LIN {X 0,Y 361.89,Z 300.406,A -85,B 0,C 180,E1 -12980.461,E2 -12980.461} C_VEL
LIN {X 0,Y 361.897,Z 300.402,A -85,B 0,C 180,E1 -12984.112,E2 -12984.112} C_VEL
LIN {X 0,Y 361.838,Z 300.409,A -85,B 0,C 180,E1 -12987.785,E2 -12987.785} C_VEL
LIN {X 0,Y 361.848,Z 300.411,A -85,B 0,C 180,E1 -12991.284,E2 -12991.284} C_VEL
LIN {X 0,Y 361.854,Z 300.407,A -85,B 0,C 180,E1 -12994.28,E2 -12994.28} C_VEL
LIN {X 0,Y 361.861,Z 300.411,A -85,B 0,C 180,E1 -12997.221,E2 -12997.221} C_VEL
LIN {X 0,Y 361.814,Z 300.414,A -85,B 0,C 180,E1 -13000.75,E2 -13000.75} C_VEL
LIN {X 0,Y 361.814,Z 300.412,A -85,B 0,C 180,E1 -13004.369,E2 -13004.369} C_VEL
LIN {X 0,Y 361.831,Z 300.414,A -85,B 0,C 180,E1 -13007.569,E2 -13007.569} C_VEL
LIN {X 0,Y 361.845,Z 300.413,A -85,B 0,C 180,E1 -13011.571,E2 -13011.571} C_VEL
LIN {X 0,Y 361.872,Z 300.405,A -85,B 0,C 180,E1 -13014.656,E2 -13014.656} C_VEL
LIN {X 0,Y 361.84,Z 300.413,A -85,B 0,C 180,E1 -13018.37,E2 -13018.37} C_VEL
LIN {X 0,Y 361.91,Z 300.458,A -85,B 0,C 180,E1 -13020.35,E2 -13020.35} C_VEL
LIN {X 0,Y 364.458,Z 313.266,A -85,B 0,C 180,E1 -13023.398,E2 -13023.398} C_VEL
LIN {X 0,Y 365.319,Z 318.996,A -85,B 0,C 180,E1 -13024.714,E2 -13024.714} C_VEL
LIN {X 0,Y 363.817,Z 337.623,A -85,B 0,C 180,E1 -13028.704,E2 -13028.704} C_VEL
LIN {X 0,Y 368.558,Z 374.157,A -85,B 0,C 180,E1 -13029.685,E2 -13029.685} C_VEL
LIN {X 0,Y 367.481,Z 446.165,A -85,B 0,C 180,E1 -13031.099,E2 -13031.099} C_VEL
LIN {X 0,Y 366.821,Z 459.565,A -85,B 0,C 180,E1 -13031.57,E2 -13031.57} C_VEL
LIN {X 0,Y 366.07,Z 472.403,A -85,B 0,C 180,E1 -13032.255,E2 -13032.255} C_VEL
LIN {X 0,Y 365.162,Z 483.779,A -85,B 0,C 180,E1 -13033.076,E2 -13033.076} C_VEL
LIN {X 0,Y 364.124,Z 495.519,A -85,B 0,C 180,E1 -13034.179,E2 -13034.179} C_VEL
LIN {X 0,Y 363.263,Z 506.09,A -85,B 0,C 180,E1 -13035.432,E2 -13035.432} C_VEL
LIN {X 0,Y 362.404,Z 515.589,A -85,B 0,C 180,E1 -13036.828,E2 -13036.828} C_VEL
LIN {X 0,Y 361.739,Z 523.371,A -85,B 0,C 180,E1 -13038.228,E2 -13038.228} C_VEL
LIN {X 0,Y 361.12,Z 530.982,A -85,B 0,C 180,E1 -13039.912,E2 -13039.912} C_VEL
LIN {X 0,Y 360.705,Z 537.097,A -85,B 0,C 180,E1 -13041.597,E2 -13041.597} C_VEL
LIN {X 0,Y 360.497,Z 541.932,A -85,B 0,C 180,E1 -13043.282,E2 -13043.282} C_VEL
LIN {X 0,Y 360.413,Z 545.63,A -85,B 0,C 180,E1 -13044.965,E2 -13044.965} C_VEL
LIN {X 0,Y 360.342,Z 548.292,A -85,B 0,C 180,E1 -13046.645,E2 -13046.645} C_VEL
LIN {X 0,Y 360.39,Z 549.547,A -85,B 0,C 180,E1 -13047.764,E2 -13047.764} C_VEL
LIN {X 0,Y 360.474,Z 550.389,A -85,B 0,C 180,E1 -13048.882,E2 -13048.882} C_VEL
LIN {X 0,Y 360.478,Z 550.79,A -85,B 0,C 180,E1 -13049.999,E2 -13049.999} C_VEL
LIN {X 0,Y 360.453,Z 550.799,A -85,B 0,C 180,E1 -13051.116,E2 -13051.116} C_VEL
LIN {X 0,Y 360.324,Z 549.647,A -85,B 0,C 180,E1 -13053.354,E2 -13053.354} C_VEL
LIN {X 0,Y 360.368,Z 548.437,A -85,B 0,C 180,E1 -13054.473,E2 -13054.473} C_VEL
LIN {X 0,Y 360.377,Z 546.224,A -85,B 0,C 180,E1 -13055.96,E2 -13055.96} C_VEL
LIN {X 0,Y 360.658,Z 542.298,A -85,B 0,C 180,E1 -13057.839,E2 -13057.839} C_VEL
LIN {X 0,Y 361.037,Z 537.639,A -85,B 0,C 180,E1 -13059.523,E2 -13059.523} C_VEL
LIN {X 0,Y 361.794,Z 530.633,A -85,B 0,C 180,E1 -13061.484,E2 -13061.484} C_VEL
LIN {X 0,Y 362.831,Z 523.079,A -85,B 0,C 180,E1 -13063.155,E2 -13063.155} C_VEL
LIN {X 0,Y 363.926,Z 513.963,A -85,B 0,C 180,E1 -13064.773,E2 -13064.773} C_VEL
LIN {X 0,Y 365.164,Z 503.913,A -85,B 0,C 180,E1 -13066.204,E2 -13066.204} C_VEL
LIN {X 0,Y 366.504,Z 493.117,A -85,B 0,C 180,E1 -13067.434,E2 -13067.434} C_VEL
LIN {X 0,Y 367.68,Z 482.609,A -85,B 0,C 180,E1 -13068.384,E2 -13068.384} C_VEL
LIN {X 0,Y 368.89,Z 469.987,A -85,B 0,C 180,E1 -13069.258,E2 -13069.258} C_VEL
LIN {X 0,Y 369.903,Z 456.623,A -85,B 0,C 180,E1 -13069.925,E2 -13069.925} C_VEL
LIN {X 0,Y 370.552,Z 444.241,A -85,B 0,C 180,E1 -13070.32,E2 -13070.32} C_VEL
LIN {X 0,Y 371.853,Z 373.551,A -85,B 0,C 180,E1 -13071.717,E2 -13071.717} C_VEL
LIN {X 0,Y 368.117,Z 350.904,A -85,B 0,C 180,E1 -13072.459,E2 -13072.459} C_VEL
LIN {X 0,Y 365.404,Z 336.978,A -85,B 0,C 180,E1 -13072.983,E2 -13072.983} C_VEL
LIN {X 0,Y 366.681,Z 324.457,A -85,B 0,C 180,E1 -13075.733,E2 -13075.733} C_VEL
LIN {X 0,Y 366.508,Z 321.277,A -85,B 0,C 180,E1 -13076.476,E2 -13076.476} C_VEL
LIN {X 0,Y 364.106,Z 309.636,A -85,B 0,C 180,E1 -13079.4,E2 -13079.4} C_VEL
LIN {X 0,Y 361.877,Z 300.409,A -85,B 0,C 180,E1 -13081.87,E2 -13081.87} C_VEL
LIN {X 0,Y 361.865,Z 300.412,A -85,B 0,C 180,E1 -13085.636,E2 -13085.636} C_VEL
LIN {X 0,Y 361.865,Z 300.407,A -85,B 0,C 180,E1 -13089.026,E2 -13089.026} C_VEL
LIN {X 0,Y 361.833,Z 300.414,A -85,B 0,C 180,E1 -13092.828,E2 -13092.828} C_VEL
LIN {X 0,Y 361.815,Z 300.415,A -85,B 0,C 180,E1 -13095.946,E2 -13095.946} C_VEL
LIN {X 0,Y 361.833,Z 300.409,A -85,B 0,C 180,E1 -13099.244,E2 -13099.244} C_VEL
LIN {X 0,Y 361.86,Z 300.409,A -85,B 0,C 180,E1 -13102.777,E2 -13102.777} C_VEL
LIN {X 0,Y 361.85,Z 300.404,A -85,B 0,C 180,E1 -13105.719,E2 -13105.719} C_VEL
LIN {X 0,Y 361.869,Z 300.404,A -85,B 0,C 180,E1 -13109.672,E2 -13109.672} C_VEL
LIN {X 0,Y 361.95,Z 300.395,A -85,B 0,C 180,E1 -13113.475,E2 -13113.475} C_VEL
LIN {X 0,Y 361.888,Z 300.405,A -85,B 0,C 180,E1 -13117.145,E2 -13117.145} C_VEL
LIN {X 0,Y 361.903,Z 300.402,A -85,B 0,C 180,E1 -13120.723,E2 -13120.723} C_VEL
LIN {X 0,Y 361.929,Z 300.396,A -85,B 0,C 180,E1 -13123.066,E2 -13123.066} C_VEL
LIN {X 0,Y 361.995,Z 300.395,A -85,B 0,C 180,E1 -13126.528,E2 -13126.528} C_VEL
LIN {X 0,Y 362.028,Z 300.387,A -85,B 0,C 180,E1 -13129.938,E2 -13129.938} C_VEL
LIN {X 0,Y 362.147,Z 300.367,A -85,B 0,C 180,E1 -13132.193,E2 -13132.193} C_VEL
LIN {X 0,Y 362.115,Z 300.378,A -85,B 0,C 180,E1 -13134.431,E2 -13134.431} C_VEL
LIN {X 0,Y 362.28,Z 300.354,A -85,B 0,C 180,E1 -13137.777,E2 -13137.777} C_VEL
LIN {X 0,Y 362.425,Z 300.333,A -85,B 0,C 180,E1 -13140,E2 -13140} C_VEL
LIN {X 0,Y 362.279,Z 300.354,A -85,B 0,C 180,E1 -13142.224,E2 -13142.224} C_VEL
LIN {X 0,Y 362.169,Z 300.37,A -85,B 0,C 180,E1 -13146.687,E2 -13146.687} C_VEL
LIN {X 0,Y 362.071,Z 300.379,A -85,B 0,C 180,E1 -13148.934,E2 -13148.934} C_VEL
LIN {X 0,Y 361.957,Z 300.395,A -85,B 0,C 180,E1 -13152.333,E2 -13152.333} C_VEL
LIN {X 0,Y 361.959,Z 300.394,A -85,B 0,C 180,E1 -13154.621,E2 -13154.621} C_VEL
LIN {X 0,Y 361.953,Z 300.393,A -85,B 0,C 180,E1 -13158.1,E2 -13158.1} C_VEL
LIN {X 0,Y 361.889,Z 300.402,A -85,B 0,C 180,E1 -13161.654,E2 -13161.654} C_VEL
LIN {X 0,Y 361.926,Z 300.398,A -85,B 0,C 180,E1 -13165.291,E2 -13165.291} C_VEL
LIN {X 0,Y 361.906,Z 300.401,A -85,B 0,C 180,E1 -13167.78,E2 -13167.78} C_VEL
LIN {X 0,Y 361.835,Z 300.408,A -85,B 0,C 180,E1 -13171.63,E2 -13171.63} C_VEL
LIN {X 0,Y 361.872,Z 300.405,A -85,B 0,C 180,E1 -13175.346,E2 -13175.346} C_VEL
LIN {X 0,Y 361.828,Z 300.41,A -85,B 0,C 180,E1 -13179.02,E2 -13179.02} C_VEL
LIN {X 0,Y 361.832,Z 300.413,A -85,B 0,C 180,E1 -13182.83,E2 -13182.83} C_VEL
LIN {X 0,Y 361.816,Z 300.415,A -85,B 0,C 180,E1 -13185.948,E2 -13185.948} C_VEL
LIN {X 0,Y 361.812,Z 300.417,A -85,B 0,C 180,E1 -13189.25,E2 -13189.25} C_VEL
LIN {X 0,Y 361.863,Z 300.409,A -85,B 0,C 180,E1 -13192.982,E2 -13192.982} C_VEL
LIN {X 0,Y 361.912,Z 300.452,A -85,B 0,C 180,E1 -13196.157,E2 -13196.157} C_VEL
LIN {X 0,Y 363.352,Z 306.792,A -85,B 0,C 180,E1 -13197.918,E2 -13197.918} C_VEL
LIN {X 0,Y 371.045,Z 324.996,A -85,B 0,C 180,E1 -13198.893,E2 -13198.893} C_VEL
LIN {X 0,Y 372.634,Z 331.878,A -85,B 0,C 180,E1 -13199.153,E2 -13199.153} C_VEL
LIN {X 0,Y 370.893,Z 414.17,A -85,B 0,C 180,E1 -13200.776,E2 -13200.776} C_VEL
LIN {X 0,Y 370.455,Z 426.98,A -85,B 0,C 180,E1 -13201.245,E2 -13201.245} C_VEL
LIN {X 0,Y 369.565,Z 439.722,A -85,B 0,C 180,E1 -13201.923,E2 -13201.923} C_VEL
LIN {X 0,Y 368.595,Z 451.32,A -85,B 0,C 180,E1 -13202.768,E2 -13202.768} C_VEL
LIN {X 0,Y 367.649,Z 461.868,A -85,B 0,C 180,E1 -13203.765,E2 -13203.765} C_VEL
LIN {X 0,Y 366.35,Z 472.689,A -85,B 0,C 180,E1 -13205.037,E2 -13205.037} C_VEL
LIN {X 0,Y 365.164,Z 482.386,A -85,B 0,C 180,E1 -13206.463,E2 -13206.463} C_VEL
LIN {X 0,Y 363.969,Z 491.187,A -85,B 0,C 180,E1 -13208.084,E2 -13208.084} C_VEL
LIN {X 0,Y 362.865,Z 499.03,A -85,B 0,C 180,E1 -13209.893,E2 -13209.893} C_VEL
LIN {X 0,Y 362.172,Z 503.997,A -85,B 0,C 180,E1 -13211.327,E2 -13211.327} C_VEL
LIN {X 0,Y 361.543,Z 508.785,A -85,B 0,C 180,E1 -13213.048,E2 -13213.048} C_VEL
LIN {X 0,Y 361.053,Z 512.416,A -85,B 0,C 180,E1 -13214.766,E2 -13214.766} C_VEL
LIN {X 0,Y 360.684,Z 515.567,A -85,B 0,C 180,E1 -13216.975,E2 -13216.975} C_VEL
LIN {X 0,Y 360.42,Z 516.954,A -85,B 0,C 180,E1 -13218.756,E2 -13218.756} C_VEL
LIN {X 0,Y 360.326,Z 517.267,A -85,B 0,C 180,E1 -13221.024,E2 -13221.024} C_VEL
LIN {X 0,Y 360.39,Z 516.84,A -85,B 0,C 180,E1 -13222.155,E2 -13222.155} C_VEL
LIN {X 0,Y 360.52,Z 515.424,A -85,B 0,C 180,E1 -13223.831,E2 -13223.831} C_VEL
LIN {X 0,Y 360.616,Z 512.064,A -85,B 0,C 180,E1 -13226.089,E2 -13226.089} C_VEL
LIN {X 0,Y 360.945,Z 508.395,A -85,B 0,C 180,E1 -13227.769,E2 -13227.769} C_VEL
LIN {X 0,Y 361.231,Z 503.636,A -85,B 0,C 180,E1 -13229.443,E2 -13229.443} C_VEL
LIN {X 0,Y 361.849,Z 497.614,A -85,B 0,C 180,E1 -13231.114,E2 -13231.114} C_VEL
LIN {X 0,Y 362.565,Z 490.143,A -85,B 0,C 180,E1 -13232.778,E2 -13232.778} C_VEL
LIN {X 0,Y 363.257,Z 482.524,A -85,B 0,C 180,E1 -13234.161,E2 -13234.161} C_VEL
LIN {X 0,Y 364.207,Z 472.185,A -85,B 0,C 180,E1 -13235.676,E2 -13235.676} C_VEL
LIN {X 0,Y 365.107,Z 461.661,A -85,B 0,C 180,E1 -13236.911,E2 -13236.911} C_VEL
LIN {X 0,Y 366.048,Z 449.853,A -85,B 0,C 180,E1 -13238.002,E2 -13238.002} C_VEL
LIN {X 0,Y 366.715,Z 437.268,A -85,B 0,C 180,E1 -13238.889,E2 -13238.889} C_VEL
LIN {X 0,Y 367.34,Z 424.615,A -85,B 0,C 180,E1 -13239.534,E2 -13239.534} C_VEL
LIN {X 0,Y 367.704,Z 411.123,A -85,B 0,C 180,E1 -13239.973,E2 -13239.973} C_VEL
LIN {X 0,Y 368.993,Z 329.473,A -85,B 0,C 180,E1 -13241.561,E2 -13241.561} C_VEL
LIN {X 0,Y 367.848,Z 322.933,A -85,B 0,C 180,E1 -13241.751,E2 -13241.751} C_VEL
LIN {X 0,Y 366.65,Z 319.026,A -85,B 0,C 180,E1 -13241.914,E2 -13241.914} C_VEL
LIN {X 0,Y 363.679,Z 314.478,A -85,B 0,C 180,E1 -13242.163,E2 -13242.163} C_VEL
LIN {X 0,Y 356.055,Z 306.492,A -85,B 0,C 180,E1 -13242.748,E2 -13242.748} C_VEL
LIN {X 0,Y 356.025,Z 306.416,A -85,B 0,C 180,E1 -13242.766,E2 -13242.766} C_VEL
LIN {X 0,Y 354.945,Z 301.27,A -85,B 0,C 180,E1 -13244.137,E2 -13244.137} C_VEL
LIN {X 0,Y 354.895,Z 301.275,A -85,B 0,C 180,E1 -13248.093,E2 -13248.093} C_VEL
LIN {X 0,Y 354.82,Z 301.284,A -85,B 0,C 180,E1 -13252.108,E2 -13252.108} C_VEL
LIN {X 0,Y 354.853,Z 301.283,A -85,B 0,C 180,E1 -13254.578,E2 -13254.578} C_VEL
LIN {X 0,Y 354.802,Z 301.287,A -85,B 0,C 180,E1 -13258.386,E2 -13258.386} C_VEL
LIN {X 0,Y 354.792,Z 301.287,A -85,B 0,C 180,E1 -13262.334,E2 -13262.334} C_VEL
LIN {X 0,Y 354.827,Z 301.283,A -85,B 0,C 180,E1 -13265.699,E2 -13265.699} C_VEL
LIN {X 0,Y 354.773,Z 301.293,A -85,B 0,C 180,E1 -13269.413,E2 -13269.413} C_VEL
LIN {X 0,Y 354.788,Z 301.29,A -85,B 0,C 180,E1 -13272.866,E2 -13272.866} C_VEL
LIN {X 0,Y 354.768,Z 301.29,A -85,B 0,C 180,E1 -13276.103,E2 -13276.103} C_VEL
LIN {X 0,Y 354.77,Z 301.294,A -85,B 0,C 180,E1 -13279.176,E2 -13279.176} C_VEL
LIN {X 0,Y 354.804,Z 301.285,A -85,B 0,C 180,E1 -13282.404,E2 -13282.404} C_VEL
LIN {X 0,Y 354.813,Z 301.285,A -85,B 0,C 180,E1 -13284.94,E2 -13284.94} C_VEL
LIN {X 0,Y 354.798,Z 301.286,A -85,B 0,C 180,E1 -13288.405,E2 -13288.405} C_VEL
LIN {X 0,Y 354.806,Z 301.291,A -85,B 0,C 180,E1 -13291.615,E2 -13291.615} C_VEL
LIN {X 0,Y 354.811,Z 301.287,A -85,B 0,C 180,E1 -13295.42,E2 -13295.42} C_VEL
LIN {X 0,Y 354.832,Z 301.282,A -85,B 0,C 180,E1 -13299.113,E2 -13299.113} C_VEL
LIN {X 0,Y 354.885,Z 301.275,A -85,B 0,C 180,E1 -13302.719,E2 -13302.719} C_VEL
LIN {X 0,Y 354.956,Z 301.27,A -85,B 0,C 180,E1 -13306.255,E2 -13306.255} C_VEL
LIN {X 0,Y 354.956,Z 301.269,A -85,B 0,C 180,E1 -13309.735,E2 -13309.735} C_VEL
LIN {X 0,Y 355.092,Z 301.249,A -85,B 0,C 180,E1 -13313.18,E2 -13313.18} C_VEL
LIN {X 0,Y 355.231,Z 301.234,A -85,B 0,C 180,E1 -13317.732,E2 -13317.732} C_VEL
LIN {X 0,Y 355.167,Z 301.24,A -85,B 0,C 180,E1 -13321.134,E2 -13321.134} C_VEL
LIN {X 0,Y 355.229,Z 301.238,A -85,B 0,C 180,E1 -13322.267,E2 -13322.267} C_VEL
LIN {X 0,Y 355.089,Z 301.252,A -85,B 0,C 180,E1 -13326.82,E2 -13326.82} C_VEL
LIN {X 0,Y 354.954,Z 301.27,A -85,B 0,C 180,E1 -13330.265,E2 -13330.265} C_VEL
LIN {X 0,Y 354.947,Z 301.269,A -85,B 0,C 180,E1 -13334.018,E2 -13334.018} C_VEL
LIN {X 0,Y 354.894,Z 301.275,A -85,B 0,C 180,E1 -13338.092,E2 -13338.092} C_VEL
LIN {X 0,Y 354.818,Z 301.284,A -85,B 0,C 180,E1 -13342.107,E2 -13342.107} C_VEL
LIN {X 0,Y 354.851,Z 301.283,A -85,B 0,C 180,E1 -13344.577,E2 -13344.577} C_VEL
LIN {X 0,Y 354.8,Z 301.287,A -85,B 0,C 180,E1 -13348.385,E2 -13348.385} C_VEL
LIN {X 0,Y 354.788,Z 301.288,A -85,B 0,C 180,E1 -13352.333,E2 -13352.333} C_VEL
LIN {X 0,Y 354.821,Z 301.284,A -85,B 0,C 180,E1 -13355.698,E2 -13355.698} C_VEL
LIN {X 0,Y 354.771,Z 301.293,A -85,B 0,C 180,E1 -13359.412,E2 -13359.412} C_VEL
LIN {X 0,Y 354.785,Z 301.29,A -85,B 0,C 180,E1 -13362.866,E2 -13362.866} C_VEL
LIN {X 0,Y 354.765,Z 301.29,A -85,B 0,C 180,E1 -13366.102,E2 -13366.102} C_VEL
LIN {X 0,Y 354.768,Z 301.294,A -85,B 0,C 180,E1 -13369.175,E2 -13369.175} C_VEL
LIN {X 0,Y 354.801,Z 301.285,A -85,B 0,C 180,E1 -13372.404,E2 -13372.404} C_VEL
LIN {X 0,Y 354.81,Z 301.286,A -85,B 0,C 180,E1 -13374.94,E2 -13374.94} C_VEL
LIN {X 0,Y 354.796,Z 301.29,A -85,B 0,C 180,E1 -13378.405,E2 -13378.405} C_VEL
LIN {X 0,Y 354.866,Z 301.367,A -85,B 0,C 180,E1 -13380.077,E2 -13380.077} C_VEL
LIN {X 0,Y 357.347,Z 313.816,A -85,B 0,C 180,E1 -13383.105,E2 -13383.105} C_VEL
LIN {X 0,Y 358.345,Z 320.219,A -85,B 0,C 180,E1 -13384.607,E2 -13384.607} C_VEL
LIN {X 0,Y 356.886,Z 337.27,A -85,B 0,C 180,E1 -13388.331,E2 -13388.331} C_VEL
LIN {X 0,Y 361.797,Z 374.503,A -85,B 0,C 180,E1 -13389.363,E2 -13389.363} C_VEL
LIN {X 0,Y 360.661,Z 446.24,A -85,B 0,C 180,E1 -13390.801,E2 -13390.801} C_VEL
LIN {X 0,Y 359.967,Z 459.5,A -85,B 0,C 180,E1 -13391.28,E2 -13391.28} C_VEL
LIN {X 0,Y 359.213,Z 472.277,A -85,B 0,C 180,E1 -13391.978,E2 -13391.978} C_VEL
LIN {X 0,Y 358.191,Z 484.392,A -85,B 0,C 180,E1 -13392.883,E2 -13392.883} C_VEL
LIN {X 0,Y 357.12,Z 495.959,A -85,B 0,C 180,E1 -13394.007,E2 -13394.007} C_VEL
LIN {X 0,Y 356.353,Z 505.318,A -85,B 0,C 180,E1 -13395.144,E2 -13395.144} C_VEL
LIN {X 0,Y 355.45,Z 514.913,A -85,B 0,C 180,E1 -13396.565,E2 -13396.565} C_VEL
LIN {X 0,Y 354.749,Z 522.762,A -85,B 0,C 180,E1 -13397.993,E2 -13397.993} C_VEL
LIN {X 0,Y 354.071,Z 530.422,A -85,B 0,C 180,E1 -13399.709,E2 -13399.709} C_VEL
LIN {X 0,Y 353.649,Z 536.582,A -85,B 0,C 180,E1 -13401.428,E2 -13401.428} C_VEL
LIN {X 0,Y 353.416,Z 541.457,A -85,B 0,C 180,E1 -13403.147,E2 -13403.147} C_VEL
LIN {X 0,Y 353.315,Z 545.192,A -85,B 0,C 180,E1 -13404.864,E2 -13404.864} C_VEL
LIN {X 0,Y 353.262,Z 547.89,A -85,B 0,C 180,E1 -13406.578,E2 -13406.578} C_VEL
LIN {X 0,Y 353.292,Z 549.16,A -85,B 0,C 180,E1 -13407.719,E2 -13407.719} C_VEL
LIN {X 0,Y 353.377,Z 550.028,A -85,B 0,C 180,E1 -13408.86,E2 -13408.86} C_VEL
LIN {X 0,Y 353.396,Z 550.451,A -85,B 0,C 180,E1 -13409.999,E2 -13409.999} C_VEL
LIN {X 0,Y 353.355,Z 550.476,A -85,B 0,C 180,E1 -13411.139,E2 -13411.139} C_VEL
LIN {X 0,Y 353.244,Z 549.362,A -85,B 0,C 180,E1 -13413.421,E2 -13413.421} C_VEL
LIN {X 0,Y 353.28,Z 548.177,A -85,B 0,C 180,E1 -13414.563,E2 -13414.563} C_VEL
LIN {X 0,Y 353.414,Z 544.561,A -85,B 0,C 180,E1 -13416.852,E2 -13416.852} C_VEL
LIN {X 0,Y 353.717,Z 540.671,A -85,B 0,C 180,E1 -13418.569,E2 -13418.569} C_VEL
LIN {X 0,Y 354.22,Z 535.668,A -85,B 0,C 180,E1 -13420.286,E2 -13420.286} C_VEL
LIN {X 0,Y 354.95,Z 529.407,A -85,B 0,C 180,E1 -13421.999,E2 -13421.999} C_VEL
LIN {X 0,Y 356.113,Z 521.614,A -85,B 0,C 180,E1 -13423.698,E2 -13423.698} C_VEL
LIN {X 0,Y 357.142,Z 513.187,A -85,B 0,C 180,E1 -13425.194,E2 -13425.194} C_VEL
LIN {X 0,Y 358.479,Z 502.962,A -85,B 0,C 180,E1 -13426.661,E2 -13426.661} C_VEL
LIN {X 0,Y 359.898,Z 491.991,A -85,B 0,C 180,E1 -13427.912,E2 -13427.912} C_VEL
LIN {X 0,Y 361.148,Z 481.265,A -85,B 0,C 180,E1 -13428.876,E2 -13428.876} C_VEL
LIN {X 0,Y 362.45,Z 468.359,A -85,B 0,C 180,E1 -13429.761,E2 -13429.761} C_VEL
LIN {X 0,Y 363.407,Z 456.035,A -85,B 0,C 180,E1 -13430.371,E2 -13430.371} C_VEL
LIN {X 0,Y 364.052,Z 443.345,A -85,B 0,C 180,E1 -13430.776,E2 -13430.776} C_VEL
LIN {X 0,Y 365.352,Z 373.939,A -85,B 0,C 180,E1 -13432.172,E2 -13432.172} C_VEL
LIN {X 0,Y 361.441,Z 350.595,A -85,B 0,C 180,E1 -13432.964,E2 -13432.964} C_VEL
LIN {X 0,Y 358.691,Z 336.589,A -85,B 0,C 180,E1 -13433.518,E2 -13433.518} C_VEL
LIN {X 0,Y 359.856,Z 324.354,A -85,B 0,C 180,E1 -13436.272,E2 -13436.272} C_VEL
LIN {X 0,Y 357.973,Z 314.576,A -85,B 0,C 180,E1 -13438.749,E2 -13438.749} C_VEL
LIN {X 0,Y 354.809,Z 301.29,A -85,B 0,C 180,E1 -13442.33,E2 -13442.33} C_VEL
LIN {X 0,Y 354.819,Z 301.29,A -85,B 0,C 180,E1 -13445.699,E2 -13445.699} C_VEL
LIN {X 0,Y 354.821,Z 301.284,A -85,B 0,C 180,E1 -13449.423,E2 -13449.423} C_VEL
LIN {X 0,Y 354.785,Z 301.292,A -85,B 0,C 180,E1 -13452.867,E2 -13452.867} C_VEL
LIN {X 0,Y 354.764,Z 301.292,A -85,B 0,C 180,E1 -13456.103,E2 -13456.103} C_VEL
LIN {X 0,Y 354.785,Z 301.287,A -85,B 0,C 180,E1 -13459.179,E2 -13459.179} C_VEL
LIN {X 0,Y 354.804,Z 301.285,A -85,B 0,C 180,E1 -13462.402,E2 -13462.402} C_VEL
LIN {X 0,Y 354.808,Z 301.283,A -85,B 0,C 180,E1 -13464.94,E2 -13464.94} C_VEL
LIN {X 0,Y 354.789,Z 301.286,A -85,B 0,C 180,E1 -13468.405,E2 -13468.405} C_VEL
LIN {X 0,Y 354.842,Z 301.277,A -85,B 0,C 180,E1 -13471.618,E2 -13471.618} C_VEL
LIN {X 0,Y 354.895,Z 301.275,A -85,B 0,C 180,E1 -13474.172,E2 -13474.172} C_VEL
LIN {X 0,Y 354.832,Z 301.282,A -85,B 0,C 180,E1 -13477.894,E2 -13477.894} C_VEL
LIN {X 0,Y 354.918,Z 301.272,A -85,B 0,C 180,E1 -13481.892,E2 -13481.892} C_VEL
LIN {X 0,Y 354.939,Z 301.27,A -85,B 0,C 180,E1 -13485.981,E2 -13485.981} C_VEL
LIN {X 0,Y 354.974,Z 301.266,A -85,B 0,C 180,E1 -13489.736,E2 -13489.736} C_VEL
LIN {X 0,Y 355.11,Z 301.243,A -85,B 0,C 180,E1 -13492.037,E2 -13492.037} C_VEL
LIN {X 0,Y 355.089,Z 301.252,A -85,B 0,C 180,E1 -13494.321,E2 -13494.321} C_VEL
LIN {X 0,Y 355.243,Z 301.231,A -85,B 0,C 180,E1 -13497.733,E2 -13497.733} C_VEL
LIN {X 0,Y 355.394,Z 301.209,A -85,B 0,C 180,E1 -13500,E2 -13500} C_VEL
LIN {X 0,Y 355.242,Z 301.231,A -85,B 0,C 180,E1 -13502.268,E2 -13502.268} C_VEL
LIN {X 0,Y 355.135,Z 301.247,A -85,B 0,C 180,E1 -13506.82,E2 -13506.82} C_VEL
LIN {X 0,Y 355.012,Z 301.258,A -85,B 0,C 180,E1 -13509.113,E2 -13509.113} C_VEL
LIN {X 0,Y 354.918,Z 301.273,A -85,B 0,C 180,E1 -13512.581,E2 -13512.581} C_VEL
LIN {X 0,Y 354.887,Z 301.275,A -85,B 0,C 180,E1 -13516.096,E2 -13516.096} C_VEL
LIN {X 0,Y 354.898,Z 301.272,A -85,B 0,C 180,E1 -13518.473,E2 -13518.473} C_VEL
LIN {X 0,Y 354.832,Z 301.281,A -85,B 0,C 180,E1 -13522.107,E2 -13522.107} C_VEL
LIN {X 0,Y 354.897,Z 301.275,A -85,B 0,C 180,E1 -13525.828,E2 -13525.828} C_VEL
LIN {X 0,Y 354.816,Z 301.287,A -85,B 0,C 180,E1 -13529.683,E2 -13529.683} C_VEL
LIN {X 0,Y 354.804,Z 301.288,A -85,B 0,C 180,E1 -13533.703,E2 -13533.703} C_VEL
LIN {X 0,Y 354.794,Z 301.286,A -85,B 0,C 180,E1 -13536.46,E2 -13536.46} C_VEL
LIN {X 0,Y 354.797,Z 301.29,A -85,B 0,C 180,E1 -13539.419,E2 -13539.419} C_VEL
LIN {X 0,Y 354.784,Z 301.291,A -85,B 0,C 180,E1 -13542.868,E2 -13542.868} C_VEL
LIN {X 0,Y 354.765,Z 301.294,A -85,B 0,C 180,E1 -13546.104,E2 -13546.104} C_VEL
LIN {X 0,Y 354.765,Z 301.295,A -85,B 0,C 180,E1 -13549.177,E2 -13549.177} C_VEL
LIN {X 0,Y 354.8,Z 301.289,A -85,B 0,C 180,E1 -13552.405,E2 -13552.405} C_VEL
LIN {X 0,Y 354.853,Z 301.46,A -85,B 0,C 180,E1 -13555.723,E2 -13555.723} C_VEL
LIN {X 0,Y 356.28,Z 307.282,A -85,B 0,C 180,E1 -13557.359,E2 -13557.359} C_VEL
LIN {X 0,Y 364.904,Z 327.394,A -85,B 0,C 180,E1 -13558.484,E2 -13558.484} C_VEL
LIN {X 0,Y 366.238,Z 333.42,A -85,B 0,C 180,E1 -13558.714,E2 -13558.714} C_VEL
LIN {X 0,Y 364.391,Z 414.619,A -85,B 0,C 180,E1 -13560.34,E2 -13560.34} C_VEL
LIN {X 0,Y 363.918,Z 427.657,A -85,B 0,C 180,E1 -13560.829,E2 -13560.829} C_VEL
LIN {X 0,Y 362.985,Z 440.431,A -85,B 0,C 180,E1 -13561.525,E2 -13561.525} C_VEL
LIN {X 0,Y 361.961,Z 451.915,A -85,B 0,C 180,E1 -13562.383,E2 -13562.383} C_VEL
LIN {X 0,Y 360.808,Z 463.7,A -85,B 0,C 180,E1 -13563.537,E2 -13563.537} C_VEL
LIN {X 0,Y 359.487,Z 474.287,A -85,B 0,C 180,E1 -13564.837,E2 -13564.837} C_VEL
LIN {X 0,Y 358.238,Z 483.691,A -85,B 0,C 180,E1 -13566.287,E2 -13566.287} C_VEL
LIN {X 0,Y 356.955,Z 492.762,A -85,B 0,C 180,E1 -13568.033,E2 -13568.033} C_VEL
LIN {X 0,Y 355.868,Z 500.003,A -85,B 0,C 180,E1 -13569.782,E2 -13569.782} C_VEL
LIN {X 0,Y 355.008,Z 505.717,A -85,B 0,C 180,E1 -13571.534,E2 -13571.534} C_VEL
LIN {X 0,Y 354.397,Z 510.179,A -85,B 0,C 180,E1 -13573.29,E2 -13573.29} C_VEL
LIN {X 0,Y 353.908,Z 513.527,A -85,B 0,C 180,E1 -13575.04,E2 -13575.04} C_VEL
LIN {X 0,Y 353.604,Z 515.944,A -85,B 0,C 180,E1 -13576.882,E2 -13576.882} C_VEL
LIN {X 0,Y 353.376,Z 517.235,A -85,B 0,C 180,E1 -13578.529,E2 -13578.529} C_VEL
LIN {X 0,Y 353.224,Z 517.617,A -85,B 0,C 180,E1 -13580.842,E2 -13580.842} C_VEL
LIN {X 0,Y 353.292,Z 517.226,A -85,B 0,C 180,E1 -13581.996,E2 -13581.996} C_VEL
LIN {X 0,Y 353.428,Z 515.718,A -85,B 0,C 180,E1 -13583.866,E2 -13583.866} C_VEL
LIN {X 0,Y 353.524,Z 512.62,A -85,B 0,C 180,E1 -13586.011,E2 -13586.011} C_VEL
LIN {X 0,Y 353.863,Z 509.025,A -85,B 0,C 180,E1 -13587.724,E2 -13587.724} C_VEL
LIN {X 0,Y 354.146,Z 504.348,A -85,B 0,C 180,E1 -13589.432,E2 -13589.432} C_VEL
LIN {X 0,Y 354.891,Z 497.306,A -85,B 0,C 180,E1 -13591.419,E2 -13591.419} C_VEL
LIN {X 0,Y 355.641,Z 489.672,A -85,B 0,C 180,E1 -13593.116,E2 -13593.116} C_VEL
LIN {X 0,Y 356.546,Z 480.102,A -85,B 0,C 180,E1 -13594.806,E2 -13594.806} C_VEL
LIN {X 0,Y 357.485,Z 470.228,A -85,B 0,C 180,E1 -13596.208,E2 -13596.208} C_VEL
LIN {X 0,Y 358.493,Z 459.067,A -85,B 0,C 180,E1 -13597.463,E2 -13597.463} C_VEL
LIN {X 0,Y 359.306,Z 448.159,A -85,B 0,C 180,E1 -13598.436,E2 -13598.436} C_VEL
LIN {X 0,Y 359.97,Z 436.117,A -85,B 0,C 180,E1 -13599.27,E2 -13599.27} C_VEL
LIN {X 0,Y 360.576,Z 423.533,A -85,B 0,C 180,E1 -13599.891,E2 -13599.891} C_VEL
LIN {X 0,Y 360.923,Z 410.379,A -85,B 0,C 180,E1 -13600.307,E2 -13600.307} C_VEL
LIN {X 0,Y 362.247,Z 330.366,A -85,B 0,C 180,E1 -13601.887,E2 -13601.887} C_VEL
LIN {X 0,Y 359.834,Z 318.307,A -85,B 0,C 180,E1 -13602.263,E2 -13602.263} C_VEL
LIN {X 0,Y 356.045,Z 306.55,A -85,B 0,C 180,E1 -13602.731,E2 -13602.731} C_VEL
LIN {X 0,Y 356.025,Z 306.416,A -85,B 0,C 180,E1 -13602.766,E2 -13602.766} C_VEL
LIN {X 0,Y 354.875,Z 304.656,A -85,B 0,C 180,E1 -13603.319,E2 -13603.319} C_VEL
LIN {X 0,Y 351.571,Z 302.922,A -85,B 0,C 180,E1 -13604.241,E2 -13604.241} C_VEL
LIN {X 0,Y 348.542,Z 302.242,A -85,B 0,C 180,E1 -13605.231,E2 -13605.231} C_VEL
LIN {X 0,Y 347.833,Z 302.154,A -85,B 0,C 180,E1 -13605.882,E2 -13605.882} C_VEL
LIN {X 0,Y 347.803,Z 302.163,A -85,B 0,C 180,E1 -13608.864,E2 -13608.864} C_VEL
LIN {X 0,Y 347.761,Z 302.166,A -85,B 0,C 180,E1 -13612.581,E2 -13612.581} C_VEL
LIN {X 0,Y 347.772,Z 302.165,A -85,B 0,C 180,E1 -13615.112,E2 -13615.112} C_VEL
LIN {X 0,Y 347.75,Z 302.17,A -85,B 0,C 180,E1 -13619.016,E2 -13619.016} C_VEL
LIN {X 0,Y 347.743,Z 302.165,A -85,B 0,C 180,E1 -13621.914,E2 -13621.914} C_VEL
LIN {X 0,Y 347.793,Z 302.159,A -85,B 0,C 180,E1 -13625.876,E2 -13625.876} C_VEL
LIN {X 0,Y 347.736,Z 302.168,A -85,B 0,C 180,E1 -13628.796,E2 -13628.796} C_VEL
LIN {X 0,Y 347.747,Z 302.165,A -85,B 0,C 180,E1 -13631.832,E2 -13631.832} C_VEL
LIN {X 0,Y 347.706,Z 302.173,A -85,B 0,C 180,E1 -13635.028,E2 -13635.028} C_VEL
LIN {X 0,Y 347.746,Z 302.164,A -85,B 0,C 180,E1 -13638.399,E2 -13638.399} C_VEL
LIN {X 0,Y 347.76,Z 302.163,A -85,B 0,C 180,E1 -13642.678,E2 -13642.678} C_VEL
LIN {X 0,Y 347.753,Z 302.166,A -85,B 0,C 180,E1 -13645.956,E2 -13645.956} C_VEL
LIN {X 0,Y 347.743,Z 302.171,A -85,B 0,C 180,E1 -13649.651,E2 -13649.651} C_VEL
LIN {X 0,Y 347.752,Z 302.169,A -85,B 0,C 180,E1 -13653.601,E2 -13653.601} C_VEL
LIN {X 0,Y 347.757,Z 302.165,A -85,B 0,C 180,E1 -13656.159,E2 -13656.159} C_VEL
LIN {X 0,Y 347.805,Z 302.163,A -85,B 0,C 180,E1 -13659.908,E2 -13659.908} C_VEL
LIN {X 0,Y 347.837,Z 302.156,A -85,B 0,C 180,E1 -13663.568,E2 -13663.568} C_VEL
LIN {X 0,Y 347.892,Z 302.146,A -85,B 0,C 180,E1 -13667.16,E2 -13667.16} C_VEL
LIN {X 0,Y 347.938,Z 302.141,A -85,B 0,C 180,E1 -13670.7,E2 -13670.7} C_VEL
LIN {X 0,Y 348.044,Z 302.133,A -85,B 0,C 180,E1 -13674.205,E2 -13674.205} C_VEL
LIN {X 0,Y 348.192,Z 302.11,A -85,B 0,C 180,E1 -13677.686,E2 -13677.686} C_VEL
LIN {X 0,Y 348.137,Z 302.116,A -85,B 0,C 180,E1 -13681.156,E2 -13681.156} C_VEL
LIN {X 0,Y 348.191,Z 302.115,A -85,B 0,C 180,E1 -13682.313,E2 -13682.313} C_VEL
LIN {X 0,Y 348.056,Z 302.127,A -85,B 0,C 180,E1 -13686.958,E2 -13686.958} C_VEL
LIN {X 0,Y 347.895,Z 302.152,A -85,B 0,C 180,E1 -13690.475,E2 -13690.475} C_VEL
LIN {X 0,Y 347.903,Z 302.147,A -85,B 0,C 180,E1 -13694.149,E2 -13694.149} C_VEL
LIN {X 0,Y 347.833,Z 302.156,A -85,B 0,C 180,E1 -13698.259,E2 -13698.259} C_VEL
LIN {X 0,Y 347.771,Z 302.161,A -85,B 0,C 180,E1 -13701.625,E2 -13701.625} C_VEL
LIN {X 0,Y 347.77,Z 302.165,A -85,B 0,C 180,E1 -13705.112,E2 -13705.112} C_VEL
LIN {X 0,Y 347.747,Z 302.17,A -85,B 0,C 180,E1 -13709.015,E2 -13709.015} C_VEL
LIN {X 0,Y 347.738,Z 302.165,A -85,B 0,C 180,E1 -13711.912,E2 -13711.912} C_VEL
LIN {X 0,Y 347.788,Z 302.159,A -85,B 0,C 180,E1 -13715.875,E2 -13715.875} C_VEL
LIN {X 0,Y 347.733,Z 302.169,A -85,B 0,C 180,E1 -13718.795,E2 -13718.795} C_VEL
LIN {X 0,Y 347.744,Z 302.166,A -85,B 0,C 180,E1 -13721.831,E2 -13721.831} C_VEL
LIN {X 0,Y 347.703,Z 302.174,A -85,B 0,C 180,E1 -13725.027,E2 -13725.027} C_VEL
LIN {X 0,Y 347.743,Z 302.165,A -85,B 0,C 180,E1 -13728.399,E2 -13728.399} C_VEL
LIN {X 0,Y 347.757,Z 302.163,A -85,B 0,C 180,E1 -13732.678,E2 -13732.678} C_VEL
LIN {X 0,Y 347.75,Z 302.166,A -85,B 0,C 180,E1 -13735.956,E2 -13735.956} C_VEL
LIN {X 0,Y 347.842,Z 302.285,A -85,B 0,C 180,E1 -13739.795,E2 -13739.795} C_VEL
LIN {X 0,Y 350.309,Z 314.53,A -85,B 0,C 180,E1 -13742.843,E2 -13742.843} C_VEL
LIN {X 0,Y 351.306,Z 320.11,A -85,B 0,C 180,E1 -13744.19,E2 -13744.19} C_VEL
LIN {X 0,Y 350.867,Z 327.062,A -85,B 0,C 180,E1 -13745.755,E2 -13745.755} C_VEL
LIN {X 0,Y 349.977,Z 336.994,A -85,B 0,C 180,E1 -13747.963,E2 -13747.963} C_VEL
LIN {X 0,Y 355.023,Z 375.735,A -85,B 0,C 180,E1 -13749.049,E2 -13749.049} C_VEL
LIN {X 0,Y 353.847,Z 446.249,A -85,B 0,C 180,E1 -13750.492,E2 -13750.492} C_VEL
LIN {X 0,Y 353.099,Z 460.166,A -85,B 0,C 180,E1 -13751.015,E2 -13751.015} C_VEL
LIN {X 0,Y 352.228,Z 473.154,A -85,B 0,C 180,E1 -13751.758,E2 -13751.758} C_VEL
LIN {X 0,Y 351.227,Z 484.979,A -85,B 0,C 180,E1 -13752.683,E2 -13752.683} C_VEL
LIN {X 0,Y 350.126,Z 496.379,A -85,B 0,C 180,E1 -13753.828,E2 -13753.828} C_VEL
LIN {X 0,Y 349.357,Z 505.199,A -85,B 0,C 180,E1 -13754.931,E2 -13754.931} C_VEL
LIN {X 0,Y 348.518,Z 514.214,A -85,B 0,C 180,E1 -13756.293,E2 -13756.293} C_VEL
LIN {X 0,Y 347.741,Z 522.134,A -85,B 0,C 180,E1 -13757.747,E2 -13757.747} C_VEL
LIN {X 0,Y 347.015,Z 529.855,A -85,B 0,C 180,E1 -13759.497,E2 -13759.497} C_VEL
LIN {X 0,Y 346.573,Z 536.061,A -85,B 0,C 180,E1 -13761.251,E2 -13761.251} C_VEL
LIN {X 0,Y 346.34,Z 540.979,A -85,B 0,C 180,E1 -13763.006,E2 -13763.006} C_VEL
LIN {X 0,Y 346.22,Z 544.751,A -85,B 0,C 180,E1 -13764.758,E2 -13764.758} C_VEL
LIN {X 0,Y 346.184,Z 547.486,A -85,B 0,C 180,E1 -13766.508,E2 -13766.508} C_VEL
LIN {X 0,Y 346.281,Z 549.661,A -85,B 0,C 180,E1 -13768.836,E2 -13768.836} C_VEL
LIN {X 0,Y 346.317,Z 550.113,A -85,B 0,C 180,E1 -13769.999,E2 -13769.999} C_VEL
LIN {X 0,Y 346.257,Z 550.153,A -85,B 0,C 180,E1 -13771.162,E2 -13771.162} C_VEL
LIN {X 0,Y 346.166,Z 549.072,A -85,B 0,C 180,E1 -13773.491,E2 -13773.491} C_VEL
LIN {X 0,Y 346.194,Z 547.92,A -85,B 0,C 180,E1 -13774.657,E2 -13774.657} C_VEL
LIN {X 0,Y 346.34,Z 544.339,A -85,B 0,C 180,E1 -13776.993,E2 -13776.993} C_VEL
LIN {X 0,Y 346.672,Z 540.487,A -85,B 0,C 180,E1 -13778.745,E2 -13778.745} C_VEL
LIN {X 0,Y 347.216,Z 535.526,A -85,B 0,C 180,E1 -13780.495,E2 -13780.495} C_VEL
LIN {X 0,Y 347.985,Z 529.31,A -85,B 0,C 180,E1 -13782.242,E2 -13782.242} C_VEL
LIN {X 0,Y 349.194,Z 521.596,A -85,B 0,C 180,E1 -13783.975,E2 -13783.975} C_VEL
LIN {X 0,Y 350.412,Z 512.019,A -85,B 0,C 180,E1 -13785.696,E2 -13785.696} C_VEL
LIN {X 0,Y 351.843,Z 502.015,A -85,B 0,C 180,E1 -13787.135,E2 -13787.135} C_VEL
LIN {X 0,Y 353.324,Z 490.841,A -85,B 0,C 180,E1 -13788.407,E2 -13788.407} C_VEL
LIN {X 0,Y 354.69,Z 479.917,A -85,B 0,C 180,E1 -13789.383,E2 -13789.383} C_VEL
LIN {X 0,Y 355.929,Z 467.856,A -85,B 0,C 180,E1 -13790.214,E2 -13790.214} C_VEL
LIN {X 0,Y 356.945,Z 455.432,A -85,B 0,C 180,E1 -13790.832,E2 -13790.832} C_VEL
LIN {X 0,Y 357.612,Z 442.557,A -85,B 0,C 180,E1 -13791.243,E2 -13791.243} C_VEL
LIN {X 0,Y 358.949,Z 375.139,A -85,B 0,C 180,E1 -13792.62,E2 -13792.62} C_VEL
LIN {X 0,Y 355.035,Z 351.733,A -85,B 0,C 180,E1 -13793.439,E2 -13793.439} C_VEL
LIN {X 0,Y 352.004,Z 336.224,A -85,B 0,C 180,E1 -13794.068,E2 -13794.068} C_VEL
LIN {X 0,Y 353.033,Z 326.136,A -85,B 0,C 180,E1 -13796.384,E2 -13796.384} C_VEL
LIN {X 0,Y 351.062,Z 315.871,A -85,B 0,C 180,E1 -13799.042,E2 -13799.042} C_VEL
LIN {X 0,Y 348.049,Z 303.477,A -85,B 0,C 180,E1 -13802.46,E2 -13802.46} C_VEL
LIN {X 0,Y 347.754,Z 302.174,A -85,B 0,C 180,E1 -13802.852,E2 -13802.852} C_VEL
LIN {X 0,Y 347.768,Z 302.169,A -85,B 0,C 180,E1 -13806.064,E2 -13806.064} C_VEL
LIN {X 0,Y 347.749,Z 302.167,A -85,B 0,C 180,E1 -13808.792,E2 -13808.792} C_VEL
LIN {X 0,Y 347.748,Z 302.165,A -85,B 0,C 180,E1 -13811.83,E2 -13811.83} C_VEL
LIN {X 0,Y 347.703,Z 302.174,A -85,B 0,C 180,E1 -13815.026,E2 -13815.026} C_VEL
LIN {X 0,Y 347.747,Z 302.167,A -85,B 0,C 180,E1 -13818.397,E2 -13818.397} C_VEL
LIN {X 0,Y 347.77,Z 302.161,A -85,B 0,C 180,E1 -13822.011,E2 -13822.011} C_VEL
LIN {X 0,Y 347.74,Z 302.162,A -85,B 0,C 180,E1 -13825.536,E2 -13825.536} C_VEL
LIN {X 0,Y 347.741,Z 302.164,A -85,B 0,C 180,E1 -13828.3,E2 -13828.3} C_VEL
LIN {X 0,Y 347.775,Z 302.16,A -85,B 0,C 180,E1 -13830.987,E2 -13830.987} C_VEL
LIN {X 0,Y 347.827,Z 302.154,A -85,B 0,C 180,E1 -13833.608,E2 -13833.608} C_VEL
LIN {X 0,Y 347.785,Z 302.155,A -85,B 0,C 180,E1 -13836.162,E2 -13836.162} C_VEL
LIN {X 0,Y 347.809,Z 302.15,A -85,B 0,C 180,E1 -13839.909,E2 -13839.909} C_VEL
LIN {X 0,Y 347.862,Z 302.154,A -85,B 0,C 180,E1 -13842.359,E2 -13842.359} C_VEL
LIN {X 0,Y 347.893,Z 302.148,A -85,B 0,C 180,E1 -13845.971,E2 -13845.971} C_VEL
LIN {X 0,Y 347.925,Z 302.144,A -85,B 0,C 180,E1 -13849.526,E2 -13849.526} C_VEL
LIN {X 0,Y 348.071,Z 302.119,A -85,B 0,C 180,E1 -13851.875,E2 -13851.875} C_VEL
LIN {X 0,Y 348.064,Z 302.127,A -85,B 0,C 180,E1 -13854.206,E2 -13854.206} C_VEL
LIN {X 0,Y 348.205,Z 302.108,A -85,B 0,C 180,E1 -13857.687,E2 -13857.687} C_VEL
LIN {X 0,Y 348.343,Z 302.088,A -85,B 0,C 180,E1 -13860,E2 -13860} C_VEL
LIN {X 0,Y 348.205,Z 302.108,A -85,B 0,C 180,E1 -13862.314,E2 -13862.314} C_VEL
LIN {X 0,Y 348.103,Z 302.125,A -85,B 0,C 180,E1 -13866.958,E2 -13866.958} C_VEL
LIN {X 0,Y 347.964,Z 302.135,A -85,B 0,C 180,E1 -13869.299,E2 -13869.299} C_VEL
LIN {X 0,Y 347.887,Z 302.147,A -85,B 0,C 180,E1 -13872.84,E2 -13872.84} C_VEL
LIN {X 0,Y 347.836,Z 302.155,A -85,B 0,C 180,E1 -13876.432,E2 -13876.432} C_VEL
LIN {X 0,Y 347.848,Z 302.153,A -85,B 0,C 180,E1 -13878.861,E2 -13878.861} C_VEL
LIN {X 0,Y 347.772,Z 302.161,A -85,B 0,C 180,E1 -13882.58,E2 -13882.58} C_VEL
LIN {X 0,Y 347.81,Z 302.157,A -85,B 0,C 180,E1 -13885.109,E2 -13885.109} C_VEL
LIN {X 0,Y 347.806,Z 302.158,A -85,B 0,C 180,E1 -13887.695,E2 -13887.695} C_VEL
LIN {X 0,Y 347.747,Z 302.165,A -85,B 0,C 180,E1 -13890.349,E2 -13890.349} C_VEL
LIN {X 0,Y 347.746,Z 302.165,A -85,B 0,C 180,E1 -13894.045,E2 -13894.045} C_VEL
LIN {X 0,Y 347.755,Z 302.166,A -85,B 0,C 180,E1 -13897.322,E2 -13897.322} C_VEL
LIN {X 0,Y 347.717,Z 302.168,A -85,B 0,C 180,E1 -13900.3,E2 -13900.3} C_VEL
LIN {X 0,Y 347.721,Z 302.17,A -85,B 0,C 180,E1 -13903.409,E2 -13903.409} C_VEL
LIN {X 0,Y 347.723,Z 302.171,A -85,B 0,C 180,E1 -13906.687,E2 -13906.687} C_VEL
LIN {X 0,Y 347.7,Z 302.175,A -85,B 0,C 180,E1 -13910.183,E2 -13910.183} C_VEL
LIN {X 0,Y 347.756,Z 302.166,A -85,B 0,C 180,E1 -13912.679,E2 -13912.679} C_VEL
LIN {X 0,Y 347.797,Z 302.178,A -85,B 0,C 180,E1 -13915.191,E2 -13915.191} C_VEL
LIN {X 0,Y 349.112,Z 307.619,A -85,B 0,C 180,E1 -13916.761,E2 -13916.761} C_VEL
LIN {X 0,Y 358.379,Z 328.876,A -85,B 0,C 180,E1 -13918.007,E2 -13918.007} C_VEL
LIN {X 0,Y 359.763,Z 334.056,A -85,B 0,C 180,E1 -13918.23,E2 -13918.23} C_VEL
LIN {X 0,Y 357.916,Z 415.134,A -85,B 0,C 180,E1 -13919.89,E2 -13919.89} C_VEL
LIN {X 0,Y 357.396,Z 428.277,A -85,B 0,C 180,E1 -13920.395,E2 -13920.395} C_VEL
LIN {X 0,Y 356.414,Z 441.134,A -85,B 0,C 180,E1 -13921.112,E2 -13921.112} C_VEL
LIN {X 0,Y 355.345,Z 452.508,A -85,B 0,C 180,E1 -13921.984,E2 -13921.984} C_VEL
LIN {X 0,Y 354.287,Z 463.066,A -85,B 0,C 180,E1 -13923.028,E2 -13923.028} C_VEL
LIN {X 0,Y 352.886,Z 473.705,A -85,B 0,C 180,E1 -13924.332,E2 -13924.332} C_VEL
LIN {X 0,Y 351.578,Z 483.328,A -85,B 0,C 180,E1 -13925.809,E2 -13925.809} C_VEL
LIN {X 0,Y 350.198,Z 492.518,A -85,B 0,C 180,E1 -13927.586,E2 -13927.586} C_VEL
LIN {X 0,Y 349.035,Z 499.874,A -85,B 0,C 180,E1 -13929.368,E2 -13929.368} C_VEL
LIN {X 0,Y 348.111,Z 505.706,A -85,B 0,C 180,E1 -13931.155,E2 -13931.155} C_VEL
LIN {X 0,Y 347.439,Z 510.25,A -85,B 0,C 180,E1 -13932.945,E2 -13932.945} C_VEL
LIN {X 0,Y 346.907,Z 513.672,A -85,B 0,C 180,E1 -13934.731,E2 -13934.731} C_VEL
LIN {X 0,Y 346.546,Z 516.309,A -85,B 0,C 180,E1 -13936.77,E2 -13936.77} C_VEL
LIN {X 0,Y 346.325,Z 517.501,A -85,B 0,C 180,E1 -13938.292,E2 -13938.292} C_VEL
LIN {X 0,Y 346.162,Z 517.937,A -85,B 0,C 180,E1 -13939.472,E2 -13939.472} C_VEL
LIN {X 0,Y 346.186,Z 517.61,A -85,B 0,C 180,E1 -13941.831,E2 -13941.831} C_VEL
LIN {X 0,Y 346.357,Z 516.042,A -85,B 0,C 180,E1 -13943.869,E2 -13943.869} C_VEL
LIN {X 0,Y 346.416,Z 514.101,A -85,B 0,C 180,E1 -13945.346,E2 -13945.346} C_VEL
LIN {X 0,Y 346.685,Z 510.919,A -85,B 0,C 180,E1 -13947.096,E2 -13947.096} C_VEL
LIN {X 0,Y 346.981,Z 506.693,A -85,B 0,C 180,E1 -13948.84,E2 -13948.84} C_VEL
LIN {X 0,Y 347.484,Z 501.291,A -85,B 0,C 180,E1 -13950.58,E2 -13950.58} C_VEL
LIN {X 0,Y 348.187,Z 494.542,A -85,B 0,C 180,E1 -13952.314,E2 -13952.314} C_VEL
LIN {X 0,Y 349.015,Z 486.153,A -85,B 0,C 180,E1 -13954.042,E2 -13954.042} C_VEL
LIN {X 0,Y 349.89,Z 477.522,A -85,B 0,C 180,E1 -13955.476,E2 -13955.476} C_VEL
LIN {X 0,Y 350.915,Z 466.903,A -85,B 0,C 180,E1 -13956.902,E2 -13956.902} C_VEL
LIN {X 0,Y 351.889,Z 456.323,A -85,B 0,C 180,E1 -13958.037,E2 -13958.037} C_VEL
LIN {X 0,Y 352.691,Z 444.525,A -85,B 0,C 180,E1 -13959.029,E2 -13959.029} C_VEL
LIN {X 0,Y 353.418,Z 432.248,A -85,B 0,C 180,E1 -13959.804,E2 -13959.804} C_VEL
LIN {X 0,Y 353.92,Z 419.637,A -85,B 0,C 180,E1 -13960.368,E2 -13960.368} C_VEL
LIN {X 0,Y 354.244,Z 404.682,A -85,B 0,C 180,E1 -13960.756,E2 -13960.756} C_VEL
LIN {X 0,Y 355.572,Z 331.714,A -85,B 0,C 180,E1 -13962.212,E2 -13962.212} C_VEL
LIN {X 0,Y 353.292,Z 320.306,A -85,B 0,C 180,E1 -13962.577,E2 -13962.577} C_VEL
LIN {X 0,Y 348.89,Z 306.851,A -85,B 0,C 180,E1 -13963.136,E2 -13963.136} C_VEL
LIN {X 0,Y 347.924,Z 302.147,A -85,B 0,C 180,E1 -13964.432,E2 -13964.432} C_VEL
LIN {X 0,Y 347.833,Z 302.154,A -85,B 0,C 180,E1 -13965.882,E2 -13965.882} C_VEL
LIN {X 0,Y 347.155,Z 302.243,A -85,B 0,C 180,E1 -13966.848,E2 -13966.848} C_VEL
LIN {X 0,Y 344.283,Z 302.602,A -85,B 0,C 180,E1 -13968.421,E2 -13968.421} C_VEL
LIN {X 0,Y 341.85,Z 302.904,A -85,B 0,C 180,E1 -13969.694,E2 -13969.694} C_VEL
LIN {X 0,Y 340.801,Z 303.035,A -85,B 0,C 180,E1 -13970.679,E2 -13970.679} C_VEL
LIN {X 0,Y 340.713,Z 303.04,A -85,B 0,C 180,E1 -13971.013,E2 -13971.013} C_VEL
LIN {X 0,Y 340.742,Z 303.042,A -85,B 0,C 180,E1 -13974.833,E2 -13974.833} C_VEL
LIN {X 0,Y 340.684,Z 303.045,A -85,B 0,C 180,E1 -13978.326,E2 -13978.326} C_VEL
LIN {X 0,Y 340.698,Z 303.049,A -85,B 0,C 180,E1 -13981.045,E2 -13981.045} C_VEL
LIN {X 0,Y 340.723,Z 303.044,A -85,B 0,C 180,E1 -13985.279,E2 -13985.279} C_VEL
LIN {X 0,Y 340.699,Z 303.043,A -85,B 0,C 180,E1 -13988.383,E2 -13988.383} C_VEL
LIN {X 0,Y 340.697,Z 303.042,A -85,B 0,C 180,E1 -13992.044,E2 -13992.044} C_VEL
LIN {X 0,Y 340.655,Z 303.047,A -85,B 0,C 180,E1 -13996.227,E2 -13996.227} C_VEL
LIN {X 0,Y 340.676,Z 303.045,A -85,B 0,C 180,E1 -13998.688,E2 -13998.688} C_VEL
LIN {X 0,Y 340.723,Z 303.042,A -85,B 0,C 180,E1 -14001.771,E2 -14001.771} C_VEL
LIN {X 0,Y 340.727,Z 303.044,A -85,B 0,C 180,E1 -14005.596,E2 -14005.596} C_VEL
LIN {X 0,Y 340.698,Z 303.043,A -85,B 0,C 180,E1 -14008.955,E2 -14008.955} C_VEL
LIN {X 0,Y 340.725,Z 303.039,A -85,B 0,C 180,E1 -14013.013,E2 -14013.013} C_VEL
LIN {X 0,Y 340.71,Z 303.04,A -85,B 0,C 180,E1 -14016.925,E2 -14016.925} C_VEL
LIN {X 0,Y 340.763,Z 303.034,A -85,B 0,C 180,E1 -14020.731,E2 -14020.731} C_VEL
LIN {X 0,Y 340.822,Z 303.027,A -85,B 0,C 180,E1 -14024.45,E2 -14024.45} C_VEL
LIN {X 0,Y 340.85,Z 303.029,A -85,B 0,C 180,E1 -14028.1,E2 -14028.1} C_VEL
LIN {X 0,Y 340.985,Z 303.009,A -85,B 0,C 180,E1 -14031.704,E2 -14031.704} C_VEL
LIN {X 0,Y 341.019,Z 303.008,A -85,B 0,C 180,E1 -14034.085,E2 -14034.085} C_VEL
LIN {X 0,Y 341.129,Z 302.989,A -85,B 0,C 180,E1 -14037.638,E2 -14037.638} C_VEL
LIN {X 0,Y 341.106,Z 302.992,A -85,B 0,C 180,E1 -14041.18,E2 -14041.18} C_VEL
LIN {X 0,Y 341.128,Z 302.995,A -85,B 0,C 180,E1 -14042.361,E2 -14042.361} C_VEL
LIN {X 0,Y 341.015,Z 303.003,A -85,B 0,C 180,E1 -14045.914,E2 -14045.914} C_VEL
LIN {X 0,Y 340.968,Z 303.013,A -85,B 0,C 180,E1 -14048.356,E2 -14048.356} C_VEL
LIN {X 0,Y 340.849,Z 303.024,A -85,B 0,C 180,E1 -14051.899,E2 -14051.899} C_VEL
LIN {X 0,Y 340.821,Z 303.027,A -85,B 0,C 180,E1 -14055.549,E2 -14055.549} C_VEL
LIN {X 0,Y 340.739,Z 303.039,A -85,B 0,C 180,E1 -14059.269,E2 -14059.269} C_VEL
LIN {X 0,Y 340.714,Z 303.044,A -85,B 0,C 180,E1 -14063.074,E2 -14063.074} C_VEL
LIN {X 0,Y 340.718,Z 303.04,A -85,B 0,C 180,E1 -14065.669,E2 -14065.669} C_VEL
LIN {X 0,Y 340.705,Z 303.042,A -85,B 0,C 180,E1 -14069.674,E2 -14069.674} C_VEL
LIN {X 0,Y 340.688,Z 303.045,A -85,B 0,C 180,E1 -14072.435,E2 -14072.435} C_VEL
LIN {X 0,Y 340.719,Z 303.044,A -85,B 0,C 180,E1 -14075.279,E2 -14075.279} C_VEL
LIN {X 0,Y 340.696,Z 303.043,A -85,B 0,C 180,E1 -14078.382,E2 -14078.382} C_VEL
LIN {X 0,Y 340.694,Z 303.043,A -85,B 0,C 180,E1 -14082.043,E2 -14082.043} C_VEL
LIN {X 0,Y 340.652,Z 303.048,A -85,B 0,C 180,E1 -14086.227,E2 -14086.227} C_VEL
LIN {X 0,Y 340.673,Z 303.046,A -85,B 0,C 180,E1 -14088.688,E2 -14088.688} C_VEL
LIN {X 0,Y 340.721,Z 303.043,A -85,B 0,C 180,E1 -14091.77,E2 -14091.77} C_VEL
LIN {X 0,Y 340.724,Z 303.045,A -85,B 0,C 180,E1 -14095.595,E2 -14095.595} C_VEL
LIN {X 0,Y 340.774,Z 303.136,A -85,B 0,C 180,E1 -14099.483,E2 -14099.483} C_VEL
LIN {X 0,Y 343.247,Z 315.241,A -85,B 0,C 180,E1 -14102.568,E2 -14102.568} C_VEL
LIN {X 0,Y 344.376,Z 322.23,A -85,B 0,C 180,E1 -14104.283,E2 -14104.283} C_VEL
LIN {X 0,Y 343.066,Z 336.651,A -85,B 0,C 180,E1 -14107.564,E2 -14107.564} C_VEL
LIN {X 0,Y 348.253,Z 375.9,A -85,B 0,C 180,E1 -14108.699,E2 -14108.699} C_VEL
LIN {X 0,Y 347.046,Z 446.259,A -85,B 0,C 180,E1 -14110.171,E2 -14110.171} C_VEL
LIN {X 0,Y 346.27,Z 460.062,A -85,B 0,C 180,E1 -14110.703,E2 -14110.703} C_VEL
LIN {X 0,Y 345.376,Z 472.973,A -85,B 0,C 180,E1 -14111.46,E2 -14111.46} C_VEL
LIN {X 0,Y 344.266,Z 485.565,A -85,B 0,C 180,E1 -14112.475,E2 -14112.475} C_VEL
LIN {X 0,Y 343.136,Z 496.794,A -85,B 0,C 180,E1 -14113.642,E2 -14113.642} C_VEL
LIN {X 0,Y 342.361,Z 505.41,A -85,B 0,C 180,E1 -14114.757,E2 -14114.757} C_VEL
LIN {X 0,Y 341.602,Z 513.502,A -85,B 0,C 180,E1 -14116.01,E2 -14116.01} C_VEL
LIN {X 0,Y 340.764,Z 521.491,A -85,B 0,C 180,E1 -14117.493,E2 -14117.493} C_VEL
LIN {X 0,Y 339.977,Z 529.283,A -85,B 0,C 180,E1 -14119.277,E2 -14119.277} C_VEL
LIN {X 0,Y 339.519,Z 535.536,A -85,B 0,C 180,E1 -14121.068,E2 -14121.068} C_VEL
LIN {X 0,Y 339.263,Z 540.496,A -85,B 0,C 180,E1 -14122.859,E2 -14122.859} C_VEL
LIN {X 0,Y 339.132,Z 544.051,A -85,B 0,C 180,E1 -14124.507,E2 -14124.507} C_VEL
LIN {X 0,Y 339.108,Z 547.079,A -85,B 0,C 180,E1 -14126.435,E2 -14126.435} C_VEL
LIN {X 0,Y 339.185,Z 549.289,A -85,B 0,C 180,E1 -14128.812,E2 -14128.812} C_VEL
LIN {X 0,Y 339.225,Z 549.774,A -85,B 0,C 180,E1 -14129.999,E2 -14129.999} C_VEL
LIN {X 0,Y 339.159,Z 549.83,A -85,B 0,C 180,E1 -14131.187,E2 -14131.187} C_VEL
LIN {X 0,Y 339.089,Z 548.784,A -85,B 0,C 180,E1 -14133.564,E2 -14133.564} C_VEL
LIN {X 0,Y 339.092,Z 547.663,A -85,B 0,C 180,E1 -14134.755,E2 -14134.755} C_VEL
LIN {X 0,Y 339.129,Z 546.097,A -85,B 0,C 180,E1 -14135.947,E2 -14135.947} C_VEL
LIN {X 0,Y 339.38,Z 542.973,A -85,B 0,C 180,E1 -14137.735,E2 -14137.735} C_VEL
LIN {X 0,Y 339.768,Z 538.804,A -85,B 0,C 180,E1 -14139.524,E2 -14139.524} C_VEL
LIN {X 0,Y 340.534,Z 532.467,A -85,B 0,C 180,E1 -14141.608,E2 -14141.608} C_VEL
LIN {X 0,Y 341.656,Z 525.596,A -85,B 0,C 180,E1 -14143.38,E2 -14143.38} C_VEL
LIN {X 0,Y 342.886,Z 517.045,A -85,B 0,C 180,E1 -14145.148,E2 -14145.148} C_VEL
LIN {X 0,Y 344.161,Z 508.289,A -85,B 0,C 180,E1 -14146.611,E2 -14146.611} C_VEL
LIN {X 0,Y 345.761,Z 497.543,A -85,B 0,C 180,E1 -14148.057,E2 -14148.057} C_VEL
LIN {X 0,Y 347.22,Z 486.83,A -85,B 0,C 180,E1 -14149.202,E2 -14149.202} C_VEL
LIN {X 0,Y 348.62,Z 474.836,A -85,B 0,C 180,E1 -14150.195,E2 -14150.195} C_VEL
LIN {X 0,Y 349.895,Z 462.347,A -85,B 0,C 180,E1 -14150.963,E2 -14150.963} C_VEL
LIN {X 0,Y 350.826,Z 449.276,A -85,B 0,C 180,E1 -14151.521,E2 -14151.521} C_VEL
LIN {X 0,Y 351.364,Z 433.583,A -85,B 0,C 180,E1 -14151.91,E2 -14151.91} C_VEL
LIN {X 0,Y 352.454,Z 375.678,A -85,B 0,C 180,E1 -14153.112,E2 -14153.112} C_VEL
LIN {X 0,Y 348.657,Z 352.718,A -85,B 0,C 180,E1 -14153.935,E2 -14153.935} C_VEL
LIN {X 0,Y 345.289,Z 336.028,A -85,B 0,C 180,E1 -14154.605,E2 -14154.605} C_VEL
LIN {X 0,Y 346.181,Z 327.817,A -85,B 0,C 180,E1 -14156.527,E2 -14156.527} C_VEL
LIN {X 0,Y 344.129,Z 317.175,A -85,B 0,C 180,E1 -14159.349,E2 -14159.349} C_VEL
LIN {X 0,Y 341.231,Z 305.217,A -85,B 0,C 180,E1 -14162.726,E2 -14162.726} C_VEL
LIN {X 0,Y 340.714,Z 303.053,A -85,B 0,C 180,E1 -14163.399,E2 -14163.399} C_VEL
LIN {X 0,Y 340.702,Z 303.048,A -85,B 0,C 180,E1 -14166.741,E2 -14166.741} C_VEL
LIN {X 0,Y 340.686,Z 303.049,A -85,B 0,C 180,E1 -14170.247,E2 -14170.247} C_VEL
LIN {X 0,Y 340.649,Z 303.052,A -85,B 0,C 180,E1 -14173.773,E2 -14173.773} C_VEL
LIN {X 0,Y 340.696,Z 303.047,A -85,B 0,C 180,E1 -14177.954,E2 -14177.954} C_VEL
LIN {X 0,Y 340.73,Z 303.038,A -85,B 0,C 180,E1 -14181.772,E2 -14181.772} C_VEL
LIN {X 0,Y 340.719,Z 303.036,A -85,B 0,C 180,E1 -14185.595,E2 -14185.595} C_VEL
LIN {X 0,Y 340.694,Z 303.042,A -85,B 0,C 180,E1 -14188.955,E2 -14188.955} C_VEL
LIN {X 0,Y 340.799,Z 303.032,A -85,B 0,C 180,E1 -14193.02,E2 -14193.02} C_VEL
LIN {X 0,Y 340.726,Z 303.042,A -85,B 0,C 180,E1 -14196.927,E2 -14196.927} C_VEL
LIN {X 0,Y 340.787,Z 303.032,A -85,B 0,C 180,E1 -14200.733,E2 -14200.733} C_VEL
LIN {X 0,Y 340.783,Z 303.028,A -85,B 0,C 180,E1 -14203.219,E2 -14203.219} C_VEL
LIN {X 0,Y 340.84,Z 303.025,A -85,B 0,C 180,E1 -14206.891,E2 -14206.891} C_VEL
LIN {X 0,Y 340.925,Z 303.019,A -85,B 0,C 180,E1 -14210.508,E2 -14210.508} C_VEL
LIN {X 0,Y 341.072,Z 302.996,A -85,B 0,C 180,E1 -14212.898,E2 -14212.898} C_VEL
LIN {X 0,Y 341.167,Z 302.985,A -85,B 0,C 180,E1 -14217.639,E2 -14217.639} C_VEL
LIN {X 0,Y 341.293,Z 302.966,A -85,B 0,C 180,E1 -14220,E2 -14220} C_VEL
LIN {X 0,Y 341.166,Z 302.985,A -85,B 0,C 180,E1 -14222.362,E2 -14222.362} C_VEL
LIN {X 0,Y 341.073,Z 303,A -85,B 0,C 180,E1 -14227.102,E2 -14227.102} C_VEL
LIN {X 0,Y 340.868,Z 303.022,A -85,B 0,C 180,E1 -14230.694,E2 -14230.694} C_VEL
LIN {X 0,Y 340.86,Z 303.02,A -85,B 0,C 180,E1 -14234.325,E2 -14234.325} C_VEL
LIN {X 0,Y 340.834,Z 303.024,A -85,B 0,C 180,E1 -14238.467,E2 -14238.467} C_VEL
LIN {X 0,Y 340.751,Z 303.035,A -85,B 0,C 180,E1 -14241.858,E2 -14241.858} C_VEL
LIN {X 0,Y 340.77,Z 303.034,A -85,B 0,C 180,E1 -14245.665,E2 -14245.665} C_VEL
LIN {X 0,Y 340.726,Z 303.039,A -85,B 0,C 180,E1 -14248.322,E2 -14248.322} C_VEL
LIN {X 0,Y 340.696,Z 303.048,A -85,B 0,C 180,E1 -14251.045,E2 -14251.045} C_VEL
LIN {X 0,Y 340.716,Z 303.039,A -85,B 0,C 180,E1 -14255.28,E2 -14255.28} C_VEL
LIN {X 0,Y 340.692,Z 303.039,A -85,B 0,C 180,E1 -14258.384,E2 -14258.384} C_VEL
LIN {X 0,Y 340.695,Z 303.046,A -85,B 0,C 180,E1 -14262.046,E2 -14262.046} C_VEL
LIN {X 0,Y 340.65,Z 303.052,A -85,B 0,C 180,E1 -14266.228,E2 -14266.228} C_VEL
LIN {X 0,Y 340.67,Z 303.05,A -85,B 0,C 180,E1 -14268.689,E2 -14268.689} C_VEL
LIN {X 0,Y 340.718,Z 303.045,A -85,B 0,C 180,E1 -14271.772,E2 -14271.772} C_VEL
LIN {X 0,Y 340.759,Z 303.083,A -85,B 0,C 180,E1 -14274.682,E2 -14274.682} C_VEL
LIN {X 0,Y 341.916,Z 307.883,A -85,B 0,C 180,E1 -14276.129,E2 -14276.129} C_VEL
LIN {X 0,Y 351.702,Z 329.978,A -85,B 0,C 180,E1 -14277.488,E2 -14277.488} C_VEL
LIN {X 0,Y 353.282,Z 334.724,A -85,B 0,C 180,E1 -14277.725,E2 -14277.725} C_VEL
LIN {X 0,Y 353.322,Z 343.74,A -85,B 0,C 180,E1 -14277.929,E2 -14277.929} C_VEL
LIN {X 0,Y 351.46,Z 415.765,A -85,B 0,C 180,E1 -14279.424,E2 -14279.424} C_VEL
LIN {X 0,Y 350.953,Z 428.287,A -85,B 0,C 180,E1 -14279.913,E2 -14279.913} C_VEL
LIN {X 0,Y 349.977,Z 440.742,A -85,B 0,C 180,E1 -14280.612,E2 -14280.612} C_VEL
LIN {X 0,Y 348.76,Z 453.134,A -85,B 0,C 180,E1 -14281.571,E2 -14281.571} C_VEL
LIN {X 0,Y 347.552,Z 464.378,A -85,B 0,C 180,E1 -14282.717,E2 -14282.717} C_VEL
LIN {X 0,Y 346.038,Z 475.304,A -85,B 0,C 180,E1 -14284.11,E2 -14284.11} C_VEL
LIN {X 0,Y 344.673,Z 484.629,A -85,B 0,C 180,E1 -14285.613,E2 -14285.613} C_VEL
LIN {X 0,Y 343.247,Z 493.65,A -85,B 0,C 180,E1 -14287.425,E2 -14287.425} C_VEL
LIN {X 0,Y 342.049,Z 500.836,A -85,B 0,C 180,E1 -14289.242,E2 -14289.242} C_VEL
LIN {X 0,Y 340.988,Z 507.072,A -85,B 0,C 180,E1 -14291.272,E2 -14291.272} C_VEL
LIN {X 0,Y 340.269,Z 511.57,A -85,B 0,C 180,E1 -14293.193,E2 -14293.193} C_VEL
LIN {X 0,Y 339.897,Z 513.804,A -85,B 0,C 180,E1 -14294.408,E2 -14294.408} C_VEL
LIN {X 0,Y 339.485,Z 516.677,A -85,B 0,C 180,E1 -14296.656,E2 -14296.656} C_VEL
LIN {X 0,Y 339.261,Z 517.752,A -85,B 0,C 180,E1 -14298.045,E2 -14298.045} C_VEL
LIN {X 0,Y 339.101,Z 518.252,A -85,B 0,C 180,E1 -14299.251,E2 -14299.251} C_VEL
LIN {X 0,Y 339.102,Z 517.992,A -85,B 0,C 180,E1 -14301.659,E2 -14301.659} C_VEL
LIN {X 0,Y 339.274,Z 516.346,A -85,B 0,C 180,E1 -14303.891,E2 -14303.891} C_VEL
LIN {X 0,Y 339.339,Z 514.616,A -85,B 0,C 180,E1 -14305.249,E2 -14305.249} C_VEL
LIN {X 0,Y 339.577,Z 511.508,A -85,B 0,C 180,E1 -14307.035,E2 -14307.035} C_VEL
LIN {X 0,Y 339.898,Z 507.357,A -85,B 0,C 180,E1 -14308.816,E2 -14308.816} C_VEL
LIN {X 0,Y 340.515,Z 501.035,A -85,B 0,C 180,E1 -14310.888,E2 -14310.888} C_VEL
LIN {X 0,Y 341.272,Z 494.152,A -85,B 0,C 180,E1 -14312.657,E2 -14312.657} C_VEL
LIN {X 0,Y 342.137,Z 485.541,A -85,B 0,C 180,E1 -14314.419,E2 -14314.419} C_VEL
LIN {X 0,Y 343.075,Z 476.721,A -85,B 0,C 180,E1 -14315.88,E2 -14315.88} C_VEL
LIN {X 0,Y 344.03,Z 467.039,A -85,B 0,C 180,E1 -14317.189,E2 -14317.189} C_VEL
LIN {X 0,Y 345.059,Z 456.401,A -85,B 0,C 180,E1 -14318.345,E2 -14318.345} C_VEL
LIN {X 0,Y 345.87,Z 444.53,A -85,B 0,C 180,E1 -14319.356,E2 -14319.356} C_VEL
LIN {X 0,Y 346.639,Z 432.148,A -85,B 0,C 180,E1 -14320.146,E2 -14320.146} C_VEL
LIN {X 0,Y 347.144,Z 419.299,A -85,B 0,C 180,E1 -14320.72,E2 -14320.72} C_VEL
LIN {X 0,Y 347.502,Z 403.84,A -85,B 0,C 180,E1 -14321.115,E2 -14321.115} C_VEL
LIN {X 0,Y 348.773,Z 332.266,A -85,B 0,C 180,E1 -14322.573,E2 -14322.573} C_VEL
LIN {X 0,Y 346.746,Z 322.231,A -85,B 0,C 180,E1 -14322.903,E2 -14322.903} C_VEL
LIN {X 0,Y 341.75,Z 307.253,A -85,B 0,C 180,E1 -14323.53,E2 -14323.53} C_VEL
LIN {X 0,Y 340.855,Z 303.029,A -85,B 0,C 180,E1 -14324.738,E2 -14324.738} C_VEL
LIN {X 0,Y 340.791,Z 303.035,A -85,B 0,C 180,E1 -14328.441,E2 -14328.441} C_VEL
LIN {X 0,Y 340.713,Z 303.04,A -85,B 0,C 180,E1 -14331.013,E2 -14331.013} C_VEL
LIN {X 0,Y 340.033,Z 303.126,A -85,B 0,C 180,E1 -14331.999,E2 -14331.999} C_VEL
LIN {X 0,Y 337.161,Z 303.483,A -85,B 0,C 180,E1 -14333.603,E2 -14333.603} C_VEL
LIN {X 0,Y 334.746,Z 303.788,A -85,B 0,C 180,E1 -14334.902,E2 -14334.902} C_VEL
LIN {X 0,Y 333.729,Z 303.91,A -85,B 0,C 180,E1 -14335.907,E2 -14335.907} C_VEL
LIN {X 0,Y 333.655,Z 303.919,A -85,B 0,C 180,E1 -14336.248,E2 -14336.248} C_VEL
LIN {X 0,Y 333.662,Z 303.92,A -85,B 0,C 180,E1 -14340.367,E2 -14340.367} C_VEL
LIN {X 0,Y 333.642,Z 303.926,A -85,B 0,C 180,E1 -14343.209,E2 -14343.209} C_VEL
LIN {X 0,Y 333.68,Z 303.917,A -85,B 0,C 180,E1 -14346.139,E2 -14346.139} C_VEL
LIN {X 0,Y 333.625,Z 303.929,A -85,B 0,C 180,E1 -14349.196,E2 -14349.196} C_VEL
LIN {X 0,Y 333.632,Z 303.922,A -85,B 0,C 180,E1 -14352.499,E2 -14352.499} C_VEL
LIN {X 0,Y 333.599,Z 303.927,A -85,B 0,C 180,E1 -14355.955,E2 -14355.955} C_VEL
LIN {X 0,Y 333.607,Z 303.93,A -85,B 0,C 180,E1 -14359.325,E2 -14359.325} C_VEL
LIN {X 0,Y 333.666,Z 303.921,A -85,B 0,C 180,E1 -14363.169,E2 -14363.169} C_VEL
LIN {X 0,Y 333.678,Z 303.92,A -85,B 0,C 180,E1 -14365.341,E2 -14365.341} C_VEL
LIN {X 0,Y 333.634,Z 303.923,A -85,B 0,C 180,E1 -14368.222,E2 -14368.222} C_VEL
LIN {X 0,Y 333.658,Z 303.92,A -85,B 0,C 180,E1 -14371.022,E2 -14371.022} C_VEL
LIN {X 0,Y 333.671,Z 303.916,A -85,B 0,C 180,E1 -14375.086,E2 -14375.086} C_VEL
LIN {X 0,Y 333.669,Z 303.918,A -85,B 0,C 180,E1 -14379.018,E2 -14379.018} C_VEL
LIN {X 0,Y 333.746,Z 303.912,A -85,B 0,C 180,E1 -14381.586,E2 -14381.586} C_VEL
LIN {X 0,Y 333.813,Z 303.9,A -85,B 0,C 180,E1 -14385.577,E2 -14385.577} C_VEL
LIN {X 0,Y 333.819,Z 303.899,A -85,B 0,C 180,E1 -14389.077,E2 -14389.077} C_VEL
LIN {X 0,Y 333.961,Z 303.882,A -85,B 0,C 180,E1 -14392.746,E2 -14392.746} C_VEL
LIN {X 0,Y 333.782,Z 303.901,A -85,B 0,C 180,E1 -14395.168,E2 -14395.168} C_VEL
LIN {X 0,Y 334.07,Z 303.868,A -85,B 0,C 180,E1 -14397.588,E2 -14397.588} C_VEL
LIN {X 0,Y 334.076,Z 303.867,A -85,B 0,C 180,E1 -14401.205,E2 -14401.205} C_VEL
LIN {X 0,Y 334.068,Z 303.873,A -85,B 0,C 180,E1 -14402.411,E2 -14402.411} C_VEL
LIN {X 0,Y 333.989,Z 303.878,A -85,B 0,C 180,E1 -14406.039,E2 -14406.039} C_VEL
LIN {X 0,Y 333.917,Z 303.892,A -85,B 0,C 180,E1 -14408.472,E2 -14408.472} C_VEL
LIN {X 0,Y 333.791,Z 303.905,A -85,B 0,C 180,E1 -14412.154,E2 -14412.154} C_VEL
LIN {X 0,Y 333.812,Z 303.906,A -85,B 0,C 180,E1 -14414.634,E2 -14414.634} C_VEL
LIN {X 0,Y 333.728,Z 303.916,A -85,B 0,C 180,E1 -14418.617,E2 -14418.617} C_VEL
LIN {X 0,Y 333.656,Z 303.921,A -85,B 0,C 180,E1 -14422.281,E2 -14422.281} C_VEL
LIN {X 0,Y 333.691,Z 303.919,A -85,B 0,C 180,E1 -14425.089,E2 -14425.089} C_VEL
LIN {X 0,Y 333.653,Z 303.926,A -85,B 0,C 180,E1 -14428.977,E2 -14428.977} C_VEL
LIN {X 0,Y 333.646,Z 303.923,A -85,B 0,C 180,E1 -14432.586,E2 -14432.586} C_VEL
LIN {X 0,Y 333.676,Z 303.918,A -85,B 0,C 180,E1 -14436.139,E2 -14436.139} C_VEL
LIN {X 0,Y 333.622,Z 303.93,A -85,B 0,C 180,E1 -14439.196,E2 -14439.196} C_VEL
LIN {X 0,Y 333.63,Z 303.924,A -85,B 0,C 180,E1 -14442.498,E2 -14442.498} C_VEL
LIN {X 0,Y 333.596,Z 303.928,A -85,B 0,C 180,E1 -14445.954,E2 -14445.954} C_VEL
LIN {X 0,Y 333.605,Z 303.931,A -85,B 0,C 180,E1 -14449.324,E2 -14449.324} C_VEL
LIN {X 0,Y 333.664,Z 303.923,A -85,B 0,C 180,E1 -14453.168,E2 -14453.168} C_VEL
LIN {X 0,Y 333.675,Z 303.923,A -85,B 0,C 180,E1 -14455.341,E2 -14455.341} C_VEL
LIN {X 0,Y 333.713,Z 303.979,A -85,B 0,C 180,E1 -14459.157,E2 -14459.157} C_VEL
LIN {X 0,Y 336.219,Z 316.131,A -85,B 0,C 180,E1 -14462.33,E2 -14462.33} C_VEL
LIN {X 0,Y 337.396,Z 323.01,A -85,B 0,C 180,E1 -14464.059,E2 -14464.059} C_VEL
LIN {X 0,Y 336.445,Z 333.984,A -85,B 0,C 180,E1 -14466.615,E2 -14466.615} C_VEL
LIN {X 0,Y 336.189,Z 336.294,A -85,B 0,C 180,E1 -14467.148,E2 -14467.148} C_VEL
LIN {X 0,Y 341.472,Z 376.041,A -85,B 0,C 180,E1 -14468.335,E2 -14468.335} C_VEL
LIN {X 0,Y 340.241,Z 445.06,A -85,B 0,C 180,E1 -14469.797,E2 -14469.797} C_VEL
LIN {X 0,Y 339.605,Z 458.416,A -85,B 0,C 180,E1 -14470.309,E2 -14470.309} C_VEL
LIN {X 0,Y 338.702,Z 470.631,A -85,B 0,C 180,E1 -14471.003,E2 -14471.003} C_VEL
LIN {X 0,Y 337.627,Z 482.954,A -85,B 0,C 180,E1 -14471.962,E2 -14471.962} C_VEL
LIN {X 0,Y 336.391,Z 494.6,A -85,B 0,C 180,E1 -14473.148,E2 -14473.148} C_VEL
LIN {X 0,Y 335.505,Z 504.319,A -85,B 0,C 180,E1 -14474.395,E2 -14474.395} C_VEL
LIN {X 0,Y 334.695,Z 512.791,A -85,B 0,C 180,E1 -14475.715,E2 -14475.715} C_VEL
LIN {X 0,Y 333.802,Z 520.841,A -85,B 0,C 180,E1 -14477.227,E2 -14477.227} C_VEL
LIN {X 0,Y 332.942,Z 528.71,A -85,B 0,C 180,E1 -14479.048,E2 -14479.048} C_VEL
LIN {X 0,Y 332.485,Z 535.012,A -85,B 0,C 180,E1 -14480.877,E2 -14480.877} C_VEL
LIN {X 0,Y 332.186,Z 540.012,A -85,B 0,C 180,E1 -14482.706,E2 -14482.706} C_VEL
LIN {X 0,Y 332.074,Z 543.069,A -85,B 0,C 180,E1 -14484.103,E2 -14484.103} C_VEL
LIN {X 0,Y 332.048,Z 544.934,A -85,B 0,C 180,E1 -14485.143,E2 -14485.143} C_VEL
LIN {X 0,Y 332.034,Z 546.672,A -85,B 0,C 180,E1 -14486.359,E2 -14486.359} C_VEL
LIN {X 0,Y 332.088,Z 548.915,A -85,B 0,C 180,E1 -14488.787,E2 -14488.787} C_VEL
LIN {X 0,Y 332.133,Z 549.432,A -85,B 0,C 180,E1 -14489.999,E2 -14489.999} C_VEL
LIN {X 0,Y 332.061,Z 549.507,A -85,B 0,C 180,E1 -14491.212,E2 -14491.212} C_VEL
LIN {X 0,Y 332.014,Z 548.495,A -85,B 0,C 180,E1 -14493.64,E2 -14493.64} C_VEL
LIN {X 0,Y 332.012,Z 546.265,A -85,B 0,C 180,E1 -14495.793,E2 -14495.793} C_VEL
LIN {X 0,Y 332.316,Z 542.772,A -85,B 0,C 180,E1 -14497.9,E2 -14497.9} C_VEL
LIN {X 0,Y 332.746,Z 538.642,A -85,B 0,C 180,E1 -14499.727,E2 -14499.727} C_VEL
LIN {X 0,Y 333.562,Z 532.351,A -85,B 0,C 180,E1 -14501.854,E2 -14501.854} C_VEL
LIN {X 0,Y 334.734,Z 525.531,A -85,B 0,C 180,E1 -14503.662,E2 -14503.662} C_VEL
LIN {X 0,Y 336.022,Z 517.07,A -85,B 0,C 180,E1 -14505.465,E2 -14505.465} C_VEL
LIN {X 0,Y 337.35,Z 508.391,A -85,B 0,C 180,E1 -14506.957,E2 -14506.957} C_VEL
LIN {X 0,Y 339.04,Z 497.732,A -85,B 0,C 180,E1 -14508.428,E2 -14508.428} C_VEL
LIN {X 0,Y 340.544,Z 487.157,A -85,B 0,C 180,E1 -14509.594,E2 -14509.594} C_VEL
LIN {X 0,Y 342,Z 475.385,A -85,B 0,C 180,E1 -14510.604,E2 -14510.604} C_VEL
LIN {X 0,Y 343.405,Z 461.877,A -85,B 0,C 180,E1 -14511.457,E2 -14511.457} C_VEL
LIN {X 0,Y 344.4,Z 448.698,A -85,B 0,C 180,E1 -14512.022,E2 -14512.022} C_VEL
LIN {X 0,Y 344.922,Z 432.886,A -85,B 0,C 180,E1 -14512.42,E2 -14512.42} C_VEL
LIN {X 0,Y 346.089,Z 376.717,A -85,B 0,C 180,E1 -14513.602,E2 -14513.602} C_VEL
LIN {X 0,Y 342.35,Z 354.031,A -85,B 0,C 180,E1 -14514.439,E2 -14514.439} C_VEL
LIN {X 0,Y 338.575,Z 335.649,A -85,B 0,C 180,E1 -14515.211,E2 -14515.211} C_VEL
LIN {X 0,Y 339.294,Z 329.141,A -85,B 0,C 180,E1 -14516.771,E2 -14516.771} C_VEL
LIN {X 0,Y 337.414,Z 319.358,A -85,B 0,C 180,E1 -14519.421,E2 -14519.421} C_VEL
LIN {X 0,Y 334.565,Z 307.527,A -85,B 0,C 180,E1 -14522.833,E2 -14522.833} C_VEL
LIN {X 0,Y 333.663,Z 303.929,A -85,B 0,C 180,E1 -14523.929,E2 -14523.929} C_VEL
LIN {X 0,Y 333.649,Z 303.924,A -85,B 0,C 180,E1 -14527.651,E2 -14527.651} C_VEL
LIN {X 0,Y 333.644,Z 303.924,A -85,B 0,C 180,E1 -14530.767,E2 -14530.767} C_VEL
LIN {X 0,Y 333.59,Z 303.933,A -85,B 0,C 180,E1 -14534.25,E2 -14534.25} C_VEL
LIN {X 0,Y 333.638,Z 303.925,A -85,B 0,C 180,E1 -14537.618,E2 -14537.618} C_VEL
LIN {X 0,Y 333.649,Z 303.921,A -85,B 0,C 180,E1 -14541.202,E2 -14541.202} C_VEL
LIN {X 0,Y 333.672,Z 303.919,A -85,B 0,C 180,E1 -14543.861,E2 -14543.861} C_VEL
LIN {X 0,Y 333.64,Z 303.921,A -85,B 0,C 180,E1 -14547.413,E2 -14547.413} C_VEL
LIN {X 0,Y 333.686,Z 303.914,A -85,B 0,C 180,E1 -14551.026,E2 -14551.026} C_VEL
LIN {X 0,Y 333.731,Z 303.91,A -85,B 0,C 180,E1 -14553.754,E2 -14553.754} C_VEL
LIN {X 0,Y 333.716,Z 303.913,A -85,B 0,C 180,E1 -14557.914,E2 -14557.914} C_VEL
LIN {X 0,Y 333.79,Z 303.905,A -85,B 0,C 180,E1 -14561.589,E2 -14561.589} C_VEL
LIN {X 0,Y 333.804,Z 303.903,A -85,B 0,C 180,E1 -14565.576,E2 -14565.576} C_VEL
LIN {X 0,Y 333.83,Z 303.902,A -85,B 0,C 180,E1 -14569.078,E2 -14569.078} C_VEL
LIN {X 0,Y 334.022,Z 303.873,A -85,B 0,C 180,E1 -14572.748,E2 -14572.748} C_VEL
LIN {X 0,Y 333.808,Z 303.9,A -85,B 0,C 180,E1 -14575.169,E2 -14575.169} C_VEL
LIN {X 0,Y 334.104,Z 303.865,A -85,B 0,C 180,E1 -14577.589,E2 -14577.589} C_VEL
LIN {X 0,Y 334.244,Z 303.844,A -85,B 0,C 180,E1 -14580,E2 -14580} C_VEL
LIN {X 0,Y 334.103,Z 303.865,A -85,B 0,C 180,E1 -14582.412,E2 -14582.412} C_VEL
LIN {X 0,Y 334.022,Z 303.877,A -85,B 0,C 180,E1 -14587.253,E2 -14587.253} C_VEL
LIN {X 0,Y 333.831,Z 303.901,A -85,B 0,C 180,E1 -14590.922,E2 -14590.922} C_VEL
LIN {X 0,Y 333.805,Z 303.901,A -85,B 0,C 180,E1 -14594.635,E2 -14594.635} C_VEL
LIN {X 0,Y 333.793,Z 303.902,A -85,B 0,C 180,E1 -14598.655,E2 -14598.655} C_VEL
LIN {X 0,Y 333.69,Z 303.914,A -85,B 0,C 180,E1 -14602.279,E2 -14602.279} C_VEL
LIN {X 0,Y 333.733,Z 303.91,A -85,B 0,C 180,E1 -14606.247,E2 -14606.247} C_VEL
LIN {X 0,Y 333.688,Z 303.915,A -85,B 0,C 180,E1 -14608.975,E2 -14608.975} C_VEL
LIN {X 0,Y 333.641,Z 303.917,A -85,B 0,C 180,E1 -14612.588,E2 -14612.588} C_VEL
LIN {X 0,Y 333.673,Z 303.917,A -85,B 0,C 180,E1 -14616.14,E2 -14616.14} C_VEL
LIN {X 0,Y 333.631,Z 303.923,A -85,B 0,C 180,E1 -14619.195,E2 -14619.195} C_VEL
LIN {X 0,Y 333.629,Z 303.926,A -85,B 0,C 180,E1 -14622.5,E2 -14622.5} C_VEL
LIN {X 0,Y 333.595,Z 303.93,A -85,B 0,C 180,E1 -14625.956,E2 -14625.956} C_VEL
LIN {X 0,Y 333.602,Z 303.93,A -85,B 0,C 180,E1 -14629.325,E2 -14629.325} C_VEL
LIN {X 0,Y 333.663,Z 303.923,A -85,B 0,C 180,E1 -14633.169,E2 -14633.169} C_VEL
LIN {X 0,Y 333.712,Z 304.039,A -85,B 0,C 180,E1 -14634.16,E2 -14634.16} C_VEL
LIN {X 0,Y 334.766,Z 308.298,A -85,B 0,C 180,E1 -14635.471,E2 -14635.471} C_VEL
LIN {X 0,Y 344.506,Z 329.698,A -85,B 0,C 180,E1 -14636.868,E2 -14636.868} C_VEL
LIN {X 0,Y 347.03,Z 336.41,A -85,B 0,C 180,E1 -14637.241,E2 -14637.241} C_VEL
LIN {X 0,Y 345.114,Z 414.757,A -85,B 0,C 180,E1 -14638.891,E2 -14638.891} C_VEL
LIN {X 0,Y 344.538,Z 427.696,A -85,B 0,C 180,E1 -14639.382,E2 -14639.382} C_VEL
LIN {X 0,Y 343.546,Z 440.338,A -85,B 0,C 180,E1 -14640.091,E2 -14640.091} C_VEL
LIN {X 0,Y 342.372,Z 452.122,A -85,B 0,C 180,E1 -14640.991,E2 -14640.991} C_VEL
LIN {X 0,Y 341.129,Z 463.231,A -85,B 0,C 180,E1 -14642.108,E2 -14642.108} C_VEL
LIN {X 0,Y 339.652,Z 473.667,A -85,B 0,C 180,E1 -14643.42,E2 -14643.42} C_VEL
LIN {X 0,Y 338.333,Z 482.519,A -85,B 0,C 180,E1 -14644.797,E2 -14644.797} C_VEL
LIN {X 0,Y 337.026,Z 490.615,A -85,B 0,C 180,E1 -14646.334,E2 -14646.334} C_VEL
LIN {X 0,Y 335.616,Z 498.471,A -85,B 0,C 180,E1 -14648.181,E2 -14648.181} C_VEL
LIN {X 0,Y 334.687,Z 503.795,A -85,B 0,C 180,E1 -14649.729,E2 -14649.729} C_VEL
LIN {X 0,Y 333.781,Z 508.913,A -85,B 0,C 180,E1 -14651.59,E2 -14651.59} C_VEL
LIN {X 0,Y 333.101,Z 512.849,A -85,B 0,C 180,E1 -14653.452,E2 -14653.452} C_VEL
LIN {X 0,Y 332.619,Z 515.719,A -85,B 0,C 180,E1 -14655.313,E2 -14655.313} C_VEL
LIN {X 0,Y 332.425,Z 517.059,A -85,B 0,C 180,E1 -14656.553,E2 -14656.553} C_VEL
LIN {X 0,Y 332.049,Z 518.551,A -85,B 0,C 180,E1 -14659.019,E2 -14659.019} C_VEL
LIN {X 0,Y 331.985,Z 518.665,A -85,B 0,C 180,E1 -14660.25,E2 -14660.25} C_VEL
LIN {X 0,Y 332.101,Z 517.698,A -85,B 0,C 180,E1 -14662.706,E2 -14662.706} C_VEL
LIN {X 0,Y 332.183,Z 516.637,A -85,B 0,C 180,E1 -14663.928,E2 -14663.928} C_VEL
LIN {X 0,Y 332.242,Z 515.133,A -85,B 0,C 180,E1 -14665.147,E2 -14665.147} C_VEL
LIN {X 0,Y 332.456,Z 512.098,A -85,B 0,C 180,E1 -14666.971,E2 -14666.971} C_VEL
LIN {X 0,Y 332.803,Z 508.022,A -85,B 0,C 180,E1 -14668.791,E2 -14668.791} C_VEL
LIN {X 0,Y 333.444,Z 501.781,A -85,B 0,C 180,E1 -14670.907,E2 -14670.907} C_VEL
LIN {X 0,Y 334.207,Z 494.994,A -85,B 0,C 180,E1 -14672.713,E2 -14672.713} C_VEL
LIN {X 0,Y 335.104,Z 486.537,A -85,B 0,C 180,E1 -14674.512,E2 -14674.512} C_VEL
LIN {X 0,Y 336.062,Z 477.848,A -85,B 0,C 180,E1 -14676.003,E2 -14676.003} C_VEL
LIN {X 0,Y 337.165,Z 467.159,A -85,B 0,C 180,E1 -14677.486,E2 -14677.486} C_VEL
LIN {X 0,Y 338.224,Z 456.455,A -85,B 0,C 180,E1 -14678.665,E2 -14678.665} C_VEL
LIN {X 0,Y 339.065,Z 444.502,A -85,B 0,C 180,E1 -14679.696,E2 -14679.696} C_VEL
LIN {X 0,Y 339.867,Z 432.004,A -85,B 0,C 180,E1 -14680.5,E2 -14680.5} C_VEL
LIN {X 0,Y 340.365,Z 419.902,A -85,B 0,C 180,E1 -14681.049,E2 -14681.049} C_VEL
LIN {X 0,Y 340.712,Z 404.644,A -85,B 0,C 180,E1 -14681.452,E2 -14681.452} C_VEL
LIN {X 0,Y 342.072,Z 333.206,A -85,B 0,C 180,E1 -14682.934,E2 -14682.934} C_VEL
LIN {X 0,Y 340.247,Z 324.275,A -85,B 0,C 180,E1 -14683.237,E2 -14683.237} C_VEL
LIN {X 0,Y 334.564,Z 307.516,A -85,B 0,C 180,E1 -14683.981,E2 -14683.981} C_VEL
LIN {X 0,Y 333.798,Z 303.905,A -85,B 0,C 180,E1 -14685.025,E2 -14685.025} C_VEL
LIN {X 0,Y 333.758,Z 303.913,A -85,B 0,C 180,E1 -14688.633,E2 -14688.633} C_VEL
LIN {X 0,Y 333.658,Z 303.921,A -85,B 0,C 180,E1 -14692.281,E2 -14692.281} C_VEL
LIN {X 0,Y 333.693,Z 303.918,A -85,B 0,C 180,E1 -14695.089,E2 -14695.089} C_VEL
LIN {X 0,Y 333.655,Z 303.919,A -85,B 0,C 180,E1 -14696.248,E2 -14696.248} C_VEL
LIN {X 0,Y 333.007,Z 304.006,A -85,B 0,C 180,E1 -14697.256,E2 -14697.256} C_VEL
LIN {X 0,Y 330.137,Z 304.366,A -85,B 0,C 180,E1 -14698.896,E2 -14698.896} C_VEL
LIN {X 0,Y 327.693,Z 304.669,A -85,B 0,C 180,E1 -14700.224,E2 -14700.224} C_VEL
LIN {X 0,Y 326.649,Z 304.796,A -85,B 0,C 180,E1 -14701.253,E2 -14701.253} C_VEL
LIN {X 0,Y 326.567,Z 304.804,A -85,B 0,C 180,E1 -14701.602,E2 -14701.602} C_VEL
LIN {X 0,Y 326.625,Z 304.802,A -85,B 0,C 180,E1 -14705.149,E2 -14705.149} C_VEL
LIN {X 0,Y 326.587,Z 304.802,A -85,B 0,C 180,E1 -14708.615,E2 -14708.615} C_VEL
LIN {X 0,Y 326.577,Z 304.804,A -85,B 0,C 180,E1 -14712.971,E2 -14712.971} C_VEL
LIN {X 0,Y 326.578,Z 304.803,A -85,B 0,C 180,E1 -14717.029,E2 -14717.029} C_VEL
LIN {X 0,Y 326.587,Z 304.806,A -85,B 0,C 180,E1 -14721.386,E2 -14721.386} C_VEL
LIN {X 0,Y 326.622,Z 304.795,A -85,B 0,C 180,E1 -14724.852,E2 -14724.852} C_VEL
LIN {X 0,Y 326.613,Z 304.8,A -85,B 0,C 180,E1 -14727.455,E2 -14727.455} C_VEL
LIN {X 0,Y 326.621,Z 304.797,A -85,B 0,C 180,E1 -14730.336,E2 -14730.336} C_VEL
LIN {X 0,Y 326.607,Z 304.794,A -85,B 0,C 180,E1 -14734.509,E2 -14734.509} C_VEL
LIN {X 0,Y 326.619,Z 304.797,A -85,B 0,C 180,E1 -14738.543,E2 -14738.543} C_VEL
LIN {X 0,Y 326.712,Z 304.785,A -85,B 0,C 180,E1 -14741.175,E2 -14741.175} C_VEL
LIN {X 0,Y 326.768,Z 304.775,A -85,B 0,C 180,E1 -14745.433,E2 -14745.433} C_VEL
LIN {X 0,Y 326.76,Z 304.779,A -85,B 0,C 180,E1 -14748.838,E2 -14748.838} C_VEL
LIN {X 0,Y 326.918,Z 304.759,A -85,B 0,C 180,E1 -14752.589,E2 -14752.589} C_VEL
LIN {X 0,Y 326.752,Z 304.776,A -85,B 0,C 180,E1 -14755.064,E2 -14755.064} C_VEL
LIN {X 0,Y 327.013,Z 304.746,A -85,B 0,C 180,E1 -14757.536,E2 -14757.536} C_VEL
LIN {X 0,Y 327.044,Z 304.743,A -85,B 0,C 180,E1 -14761.231,E2 -14761.231} C_VEL
LIN {X 0,Y 326.751,Z 304.78,A -85,B 0,C 180,E1 -14763.699,E2 -14763.699} C_VEL
LIN {X 0,Y 326.944,Z 304.756,A -85,B 0,C 180,E1 -14766.17,E2 -14766.17} C_VEL
LIN {X 0,Y 326.785,Z 304.776,A -85,B 0,C 180,E1 -14769.907,E2 -14769.907} C_VEL
LIN {X 0,Y 326.762,Z 304.778,A -85,B 0,C 180,E1 -14773.685,E2 -14773.685} C_VEL
LIN {X 0,Y 326.667,Z 304.79,A -85,B 0,C 180,E1 -14777.529,E2 -14777.529} C_VEL
LIN {X 0,Y 326.618,Z 304.797,A -85,B 0,C 180,E1 -14781.456,E2 -14781.456} C_VEL
LIN {X 0,Y 326.636,Z 304.795,A -85,B 0,C 180,E1 -14785.488,E2 -14785.488} C_VEL
LIN {X 0,Y 326.591,Z 304.801,A -85,B 0,C 180,E1 -14789.666,E2 -14789.666} C_VEL
LIN {X 0,Y 326.62,Z 304.802,A -85,B 0,C 180,E1 -14792.945,E2 -14792.945} C_VEL
LIN {X 0,Y 326.613,Z 304.799,A -85,B 0,C 180,E1 -14795.519,E2 -14795.519} C_VEL
LIN {X 0,Y 326.59,Z 304.806,A -85,B 0,C 180,E1 -14799.221,E2 -14799.221} C_VEL
LIN {X 0,Y 326.575,Z 304.806,A -85,B 0,C 180,E1 -14802.971,E2 -14802.971} C_VEL
LIN {X 0,Y 326.575,Z 304.805,A -85,B 0,C 180,E1 -14807.028,E2 -14807.028} C_VEL
LIN {X 0,Y 326.584,Z 304.807,A -85,B 0,C 180,E1 -14811.385,E2 -14811.385} C_VEL
LIN {X 0,Y 326.62,Z 304.798,A -85,B 0,C 180,E1 -14814.851,E2 -14814.851} C_VEL
LIN {X 0,Y 326.637,Z 304.837,A -85,B 0,C 180,E1 -14818.819,E2 -14818.819} C_VEL
LIN {X 0,Y 329.09,Z 316.627,A -85,B 0,C 180,E1 -14821.976,E2 -14821.976} C_VEL
LIN {X 0,Y 330.369,Z 323.706,A -85,B 0,C 180,E1 -14823.805,E2 -14823.805} C_VEL
LIN {X 0,Y 330.03,Z 329.221,A -85,B 0,C 180,E1 -14825.128,E2 -14825.128} C_VEL
LIN {X 0,Y 329.32,Z 336.042,A -85,B 0,C 180,E1 -14826.732,E2 -14826.732} C_VEL
LIN {X 0,Y 334.501,Z 374.86,A -85,B 0,C 180,E1 -14827.917,E2 -14827.917} C_VEL
LIN {X 0,Y 334.693,Z 382.192,A -85,B 0,C 180,E1 -14828.091,E2 -14828.091} C_VEL
LIN {X 0,Y 333.463,Z 444.975,A -85,B 0,C 180,E1 -14829.448,E2 -14829.448} C_VEL
LIN {X 0,Y 332.806,Z 458.25,A -85,B 0,C 180,E1 -14829.97,E2 -14829.97} C_VEL
LIN {X 0,Y 331.866,Z 470.421,A -85,B 0,C 180,E1 -14830.676,E2 -14830.676} C_VEL
LIN {X 0,Y 330.791,Z 481.893,A -85,B 0,C 180,E1 -14831.576,E2 -14831.576} C_VEL
LIN {X 0,Y 329.612,Z 493.695,A -85,B 0,C 180,E1 -14832.791,E2 -14832.791} C_VEL
LIN {X 0,Y 328.569,Z 504.113,A -85,B 0,C 180,E1 -14834.145,E2 -14834.145} C_VEL
LIN {X 0,Y 327.548,Z 513.841,A -85,B 0,C 180,E1 -14835.714,E2 -14835.714} C_VEL
LIN {X 0,Y 326.502,Z 523.012,A -85,B 0,C 180,E1 -14837.569,E2 -14837.569} C_VEL
LIN {X 0,Y 325.763,Z 530.4,A -85,B 0,C 180,E1 -14839.433,E2 -14839.433} C_VEL
LIN {X 0,Y 325.302,Z 536.317,A -85,B 0,C 180,E1 -14841.301,E2 -14841.301} C_VEL
LIN {X 0,Y 325.051,Z 540.967,A -85,B 0,C 180,E1 -14843.17,E2 -14843.17} C_VEL
LIN {X 0,Y 324.954,Z 544.494,A -85,B 0,C 180,E1 -14845.036,E2 -14845.036} C_VEL
LIN {X 0,Y 324.961,Z 546.264,A -85,B 0,C 180,E1 -14846.279,E2 -14846.279} C_VEL
LIN {X 0,Y 324.992,Z 548.542,A -85,B 0,C 180,E1 -14848.76,E2 -14848.76} C_VEL
LIN {X 0,Y 325.04,Z 549.085,A -85,B 0,C 180,E1 -14849.999,E2 -14849.999} C_VEL
LIN {X 0,Y 324.964,Z 549.185,A -85,B 0,C 180,E1 -14851.238,E2 -14851.238} C_VEL
LIN {X 0,Y 324.938,Z 548.207,A -85,B 0,C 180,E1 -14853.72,E2 -14853.72} C_VEL
LIN {X 0,Y 324.919,Z 546.226,A -85,B 0,C 180,E1 -14855.742,E2 -14855.742} C_VEL
LIN {X 0,Y 325.243,Z 542.576,A -85,B 0,C 180,E1 -14858.073,E2 -14858.073} C_VEL
LIN {X 0,Y 325.72,Z 538.489,A -85,B 0,C 180,E1 -14859.939,E2 -14859.939} C_VEL
LIN {X 0,Y 326.598,Z 532.242,A -85,B 0,C 180,E1 -14862.11,E2 -14862.11} C_VEL
LIN {X 0,Y 327.83,Z 525.472,A -85,B 0,C 180,E1 -14863.955,E2 -14863.955} C_VEL
LIN {X 0,Y 329.173,Z 517.094,A -85,B 0,C 180,E1 -14865.796,E2 -14865.796} C_VEL
LIN {X 0,Y 330.55,Z 508.492,A -85,B 0,C 180,E1 -14867.316,E2 -14867.316} C_VEL
LIN {X 0,Y 332.328,Z 497.92,A -85,B 0,C 180,E1 -14868.814,E2 -14868.814} C_VEL
LIN {X 0,Y 333.88,Z 487.458,A -85,B 0,C 180,E1 -14870.001,E2 -14870.001} C_VEL
LIN {X 0,Y 335.402,Z 475.933,A -85,B 0,C 180,E1 -14871.028,E2 -14871.028} C_VEL
LIN {X 0,Y 336.762,Z 463.986,A -85,B 0,C 180,E1 -14871.822,E2 -14871.822} C_VEL
LIN {X 0,Y 337.776,Z 451.102,A -85,B 0,C 180,E1 -14872.437,E2 -14872.437} C_VEL
LIN {X 0,Y 338.444,Z 437.443,A -85,B 0,C 180,E1 -14872.833,E2 -14872.833} C_VEL
LIN {X 0,Y 339.756,Z 377.735,A -85,B 0,C 180,E1 -14874.111,E2 -14874.111} C_VEL
LIN {X 0,Y 335.985,Z 355.01,A -85,B 0,C 180,E1 -14874.98,E2 -14874.98} C_VEL
LIN {X 0,Y 332.255,Z 337.018,A -85,B 0,C 180,E1 -14875.757,E2 -14875.757} C_VEL
LIN {X 0,Y 331.967,Z 335.249,A -85,B 0,C 180,E1 -14875.844,E2 -14875.844} C_VEL
LIN {X 0,Y 332.44,Z 331.231,A -85,B 0,C 180,E1 -14876.826,E2 -14876.826} C_VEL
LIN {X 0,Y 330.751,Z 321.881,A -85,B 0,C 180,E1 -14879.403,E2 -14879.403} C_VEL
LIN {X 0,Y 327.888,Z 309.882,A -85,B 0,C 180,E1 -14882.934,E2 -14882.934} C_VEL
LIN {X 0,Y 326.64,Z 304.805,A -85,B 0,C 180,E1 -14884.527,E2 -14884.527} C_VEL
LIN {X 0,Y 326.621,Z 304.801,A -85,B 0,C 180,E1 -14888.608,E2 -14888.608} C_VEL
LIN {X 0,Y 326.573,Z 304.802,A -85,B 0,C 180,E1 -14891.845,E2 -14891.845} C_VEL
LIN {X 0,Y 326.524,Z 304.811,A -85,B 0,C 180,E1 -14895.257,E2 -14895.257} C_VEL
LIN {X 0,Y 326.574,Z 304.801,A -85,B 0,C 180,E1 -14898.868,E2 -14898.868} C_VEL
LIN {X 0,Y 326.624,Z 304.797,A -85,B 0,C 180,E1 -14902.761,E2 -14902.761} C_VEL
LIN {X 0,Y 326.603,Z 304.796,A -85,B 0,C 180,E1 -14905.98,E2 -14905.98} C_VEL
LIN {X 0,Y 326.644,Z 304.795,A -85,B 0,C 180,E1 -14910.339,E2 -14910.339} C_VEL
LIN {X 0,Y 326.686,Z 304.79,A -85,B 0,C 180,E1 -14914.516,E2 -14914.516} C_VEL
LIN {X 0,Y 326.642,Z 304.795,A -85,B 0,C 180,E1 -14918.545,E2 -14918.545} C_VEL
LIN {X 0,Y 326.74,Z 304.785,A -85,B 0,C 180,E1 -14921.177,E2 -14921.177} C_VEL
LIN {X 0,Y 326.759,Z 304.782,A -85,B 0,C 180,E1 -14925.433,E2 -14925.433} C_VEL
LIN {X 0,Y 326.766,Z 304.779,A -85,B 0,C 180,E1 -14928.839,E2 -14928.839} C_VEL
LIN {X 0,Y 326.976,Z 304.749,A -85,B 0,C 180,E1 -14932.591,E2 -14932.591} C_VEL
LIN {X 0,Y 326.775,Z 304.777,A -85,B 0,C 180,E1 -14935.065,E2 -14935.065} C_VEL
LIN {X 0,Y 327.045,Z 304.745,A -85,B 0,C 180,E1 -14937.537,E2 -14937.537} C_VEL
LIN {X 0,Y 327.195,Z 304.722,A -85,B 0,C 180,E1 -14940,E2 -14940} C_VEL
LIN {X 0,Y 327.044,Z 304.745,A -85,B 0,C 180,E1 -14942.464,E2 -14942.464} C_VEL
LIN {X 0,Y 326.968,Z 304.75,A -85,B 0,C 180,E1 -14946.665,E2 -14946.665} C_VEL
LIN {X 0,Y 326.811,Z 304.77,A -85,B 0,C 180,E1 -14949.907,E2 -14949.907} C_VEL
LIN {X 0,Y 326.756,Z 304.777,A -85,B 0,C 180,E1 -14953.686,E2 -14953.686} C_VEL
LIN {X 0,Y 326.696,Z 304.784,A -85,B 0,C 180,E1 -14957.529,E2 -14957.529} C_VEL
LIN {X 0,Y 326.66,Z 304.792,A -85,B 0,C 180,E1 -14960.136,E2 -14960.136} C_VEL
LIN {X 0,Y 326.649,Z 304.793,A -85,B 0,C 180,E1 -14964.13,E2 -14964.13} C_VEL
LIN {X 0,Y 326.68,Z 304.792,A -85,B 0,C 180,E1 -14966.859,E2 -14966.859} C_VEL
LIN {X 0,Y 326.632,Z 304.797,A -85,B 0,C 180,E1 -14970.61,E2 -14970.61} C_VEL
LIN {X 0,Y 326.605,Z 304.799,A -85,B 0,C 180,E1 -14974.02,E2 -14974.02} C_VEL
LIN {X 0,Y 326.622,Z 304.799,A -85,B 0,C 180,E1 -14977.238,E2 -14977.238} C_VEL
LIN {X 0,Y 326.572,Z 304.802,A -85,B 0,C 180,E1 -14981.131,E2 -14981.131} C_VEL
LIN {X 0,Y 326.526,Z 304.812,A -85,B 0,C 180,E1 -14984.744,E2 -14984.744} C_VEL
LIN {X 0,Y 326.562,Z 304.807,A -85,B 0,C 180,E1 -14988.153,E2 -14988.153} C_VEL
LIN {X 0,Y 326.567,Z 304.806,A -85,B 0,C 180,E1 -14991.384,E2 -14991.384} C_VEL
LIN {X 0,Y 326.668,Z 304.916,A -85,B 0,C 180,E1 -14993.584,E2 -14993.584} C_VEL
LIN {X 0,Y 327.639,Z 308.738,A -85,B 0,C 180,E1 -14994.783,E2 -14994.783} C_VEL
LIN {X 0,Y 336.714,Z 328.266,A -85,B 0,C 180,E1 -14996.133,E2 -14996.133} C_VEL
LIN {X 0,Y 340.815,Z 338.056,A -85,B 0,C 180,E1 -14996.737,E2 -14996.737} C_VEL
LIN {X 0,Y 338.678,Z 416.011,A -85,B 0,C 180,E1 -14998.406,E2 -14998.406} C_VEL
LIN {X 0,Y 338.041,Z 429.401,A -85,B 0,C 180,E1 -14998.946,E2 -14998.946} C_VEL
LIN {X 0,Y 336.952,Z 442.249,A -85,B 0,C 180,E1 -14999.703,E2 -14999.703} C_VEL
LIN {X 0,Y 335.637,Z 454.392,A -85,B 0,C 180,E1 -15000.696,E2 -15000.696} C_VEL
LIN {X 0,Y 334.308,Z 465.569,A -85,B 0,C 180,E1 -15001.888,E2 -15001.888} C_VEL
LIN {X 0,Y 332.663,Z 476.338,A -85,B 0,C 180,E1 -15003.325,E2 -15003.325} C_VEL
LIN {X 0,Y 331.17,Z 485.595,A -85,B 0,C 180,E1 -15004.886,E2 -15004.886} C_VEL
LIN {X 0,Y 329.745,Z 493.685,A -85,B 0,C 180,E1 -15006.566,E2 -15006.566} C_VEL
LIN {X 0,Y 328.429,Z 500.602,A -85,B 0,C 180,E1 -15008.339,E2 -15008.339} C_VEL
LIN {X 0,Y 327.515,Z 505.585,A -85,B 0,C 180,E1 -15009.921,E2 -15009.921} C_VEL
LIN {X 0,Y 326.62,Z 510.386,A -85,B 0,C 180,E1 -15011.821,E2 -15011.821} C_VEL
LIN {X 0,Y 325.952,Z 514.031,A -85,B 0,C 180,E1 -15013.723,E2 -15013.723} C_VEL
LIN {X 0,Y 325.625,Z 515.896,A -85,B 0,C 180,E1 -15014.99,E2 -15014.99} C_VEL
LIN {X 0,Y 325.38,Z 517.408,A -85,B 0,C 180,E1 -15016.406,E2 -15016.406} C_VEL
LIN {X 0,Y 325.004,Z 518.835,A -85,B 0,C 180,E1 -15018.778,E2 -15018.778} C_VEL
LIN {X 0,Y 324.896,Z 519.014,A -85,B 0,C 180,E1 -15020.035,E2 -15020.035} C_VEL
LIN {X 0,Y 324.92,Z 518.757,A -85,B 0,C 180,E1 -15021.292,E2 -15021.292} C_VEL
LIN {X 0,Y 324.986,Z 518.114,A -85,B 0,C 180,E1 -15022.545,E2 -15022.545} C_VEL
LIN {X 0,Y 325.101,Z 516.937,A -85,B 0,C 180,E1 -15023.953,E2 -15023.953} C_VEL
LIN {X 0,Y 325.226,Z 513.759,A -85,B 0,C 180,E1 -15026.284,E2 -15026.284} C_VEL
LIN {X 0,Y 325.602,Z 510.104,A -85,B 0,C 180,E1 -15028.145,E2 -15028.145} C_VEL
LIN {X 0,Y 325.983,Z 505.358,A -85,B 0,C 180,E1 -15030.001,E2 -15030.001} C_VEL
LIN {X 0,Y 326.862,Z 498.241,A -85,B 0,C 180,E1 -15032.157,E2 -15032.157} C_VEL
LIN {X 0,Y 327.766,Z 490.477,A -85,B 0,C 180,E1 -15033.997,E2 -15033.997} C_VEL
LIN {X 0,Y 328.804,Z 480.807,A -85,B 0,C 180,E1 -15035.828,E2 -15035.828} C_VEL
LIN {X 0,Y 329.964,Z 470.76,A -85,B 0,C 180,E1 -15037.343,E2 -15037.343} C_VEL
LIN {X 0,Y 331.104,Z 459.393,A -85,B 0,C 180,E1 -15038.699,E2 -15038.699} C_VEL
LIN {X 0,Y 332.022,Z 448.255,A -85,B 0,C 180,E1 -15039.75,E2 -15039.75} C_VEL
LIN {X 0,Y 332.813,Z 435.744,A -85,B 0,C 180,E1 -15040.649,E2 -15040.649} C_VEL
LIN {X 0,Y 333.519,Z 422.313,A -85,B 0,C 180,E1 -15041.318,E2 -15041.318} C_VEL
LIN {X 0,Y 333.872,Z 408.961,A -85,B 0,C 180,E1 -15041.729,E2 -15041.729} C_VEL
LIN {X 0,Y 335.402,Z 334.382,A -85,B 0,C 180,E1 -15043.302,E2 -15043.302} C_VEL
LIN {X 0,Y 333.818,Z 326.591,A -85,B 0,C 180,E1 -15043.573,E2 -15043.573} C_VEL
LIN {X 0,Y 328.037,Z 309.847,A -85,B 0,C 180,E1 -15044.318,E2 -15044.318} C_VEL
LIN {X 0,Y 327.382,Z 307.744,A -85,B 0,C 180,E1 -15044.462,E2 -15044.462} C_VEL
LIN {X 0,Y 326.741,Z 304.783,A -85,B 0,C 180,E1 -15045.358,E2 -15045.358} C_VEL
LIN {X 0,Y 326.712,Z 304.79,A -85,B 0,C 180,E1 -15048.825,E2 -15048.825} C_VEL
LIN {X 0,Y 326.602,Z 304.803,A -85,B 0,C 180,E1 -15052.789,E2 -15052.789} C_VEL
LIN {X 0,Y 326.601,Z 304.798,A -85,B 0,C 180,E1 -15056.245,E2 -15056.245} C_VEL
LIN {X 0,Y 326.62,Z 304.797,A -85,B 0,C 180,E1 -15059.664,E2 -15059.664} C_VEL
LIN {X 0,Y 326.567,Z 304.804,A -85,B 0,C 180,E1 -15061.602,E2 -15061.602} C_VEL
LIN {X 0,Y 325.909,Z 304.889,A -85,B 0,C 180,E1 -15062.632,E2 -15062.632} C_VEL
LIN {X 0,Y 323.067,Z 305.239,A -85,B 0,C 180,E1 -15064.309,E2 -15064.309} C_VEL
LIN {X 0,Y 320.654,Z 305.541,A -85,B 0,C 180,E1 -15065.667,E2 -15065.667} C_VEL
LIN {X 0,Y 319.621,Z 305.671,A -85,B 0,C 180,E1 -15066.719,E2 -15066.719} C_VEL
LIN {X 0,Y 319.538,Z 305.678,A -85,B 0,C 180,E1 -15067.075,E2 -15067.075} C_VEL
LIN {X 0,Y 319.533,Z 305.68,A -85,B 0,C 180,E1 -15069.662,E2 -15069.662} C_VEL
LIN {X 0,Y 319.524,Z 305.684,A -85,B 0,C 180,E1 -15073.46,E2 -15073.46} C_VEL
LIN {X 0,Y 319.556,Z 305.677,A -85,B 0,C 180,E1 -15077.016,E2 -15077.016} C_VEL
LIN {X 0,Y 319.519,Z 305.68,A -85,B 0,C 180,E1 -15080.366,E2 -15080.366} C_VEL
LIN {X 0,Y 319.56,Z 305.678,A -85,B 0,C 180,E1 -15083.572,E2 -15083.572} C_VEL
LIN {X 0,Y 319.582,Z 305.671,A -85,B 0,C 180,E1 -15086.687,E2 -15086.687} C_VEL
LIN {X 0,Y 319.565,Z 305.681,A -85,B 0,C 180,E1 -15089.613,E2 -15089.613} C_VEL
LIN {X 0,Y 319.545,Z 305.676,A -85,B 0,C 180,E1 -15092.492,E2 -15092.492} C_VEL
LIN {X 0,Y 319.554,Z 305.673,A -85,B 0,C 180,E1 -15095.299,E2 -15095.299} C_VEL
LIN {X 0,Y 319.57,Z 305.678,A -85,B 0,C 180,E1 -15098.045,E2 -15098.045} C_VEL
LIN {X 0,Y 319.629,Z 305.669,A -85,B 0,C 180,E1 -15102.071,E2 -15102.071} C_VEL
LIN {X 0,Y 319.737,Z 305.655,A -85,B 0,C 180,E1 -15106.008,E2 -15106.008} C_VEL
LIN {X 0,Y 319.739,Z 305.657,A -85,B 0,C 180,E1 -15109.872,E2 -15109.872} C_VEL
LIN {X 0,Y 319.904,Z 305.633,A -85,B 0,C 180,E1 -15113.693,E2 -15113.693} C_VEL
LIN {X 0,Y 319.959,Z 305.624,A -85,B 0,C 180,E1 -15117.482,E2 -15117.482} C_VEL
LIN {X 0,Y 320.012,Z 305.619,A -85,B 0,C 180,E1 -15121.258,E2 -15121.258} C_VEL
LIN {X 0,Y 319.718,Z 305.653,A -85,B 0,C 180,E1 -15125.044,E2 -15125.044} C_VEL
LIN {X 0,Y 319.856,Z 305.636,A -85,B 0,C 180,E1 -15127.575,E2 -15127.575} C_VEL
LIN {X 0,Y 319.716,Z 305.657,A -85,B 0,C 180,E1 -15131.41,E2 -15131.41} C_VEL
LIN {X 0,Y 319.716,Z 305.662,A -85,B 0,C 180,E1 -15134.71,E2 -15134.71} C_VEL
LIN {X 0,Y 319.618,Z 305.669,A -85,B 0,C 180,E1 -15137.929,E2 -15137.929} C_VEL
LIN {X 0,Y 319.569,Z 305.675,A -85,B 0,C 180,E1 -15141.954,E2 -15141.954} C_VEL
LIN {X 0,Y 319.57,Z 305.675,A -85,B 0,C 180,E1 -15146.094,E2 -15146.094} C_VEL
LIN {X 0,Y 319.533,Z 305.686,A -85,B 0,C 180,E1 -15148.939,E2 -15148.939} C_VEL
LIN {X 0,Y 319.526,Z 305.681,A -85,B 0,C 180,E1 -15151.862,E2 -15151.862} C_VEL
LIN {X 0,Y 319.581,Z 305.675,A -85,B 0,C 180,E1 -15155.542,E2 -15155.542} C_VEL
LIN {X 0,Y 319.531,Z 305.681,A -85,B 0,C 180,E1 -15159.661,E2 -15159.661} C_VEL
LIN {X 0,Y 319.521,Z 305.685,A -85,B 0,C 180,E1 -15163.459,E2 -15163.459} C_VEL
LIN {X 0,Y 319.554,Z 305.679,A -85,B 0,C 180,E1 -15167.015,E2 -15167.015} C_VEL
LIN {X 0,Y 319.547,Z 305.678,A -85,B 0,C 180,E1 -15170.37,E2 -15170.37} C_VEL
LIN {X 0,Y 319.58,Z 305.675,A -85,B 0,C 180,E1 -15174.457,E2 -15174.457} C_VEL
LIN {X 0,Y 319.606,Z 305.731,A -85,B 0,C 180,E1 -15178.48,E2 -15178.48} C_VEL
LIN {X 0,Y 322.018,Z 317.32,A -85,B 0,C 180,E1 -15181.66,E2 -15181.66} C_VEL
LIN {X 0,Y 323.466,Z 325.948,A -85,B 0,C 180,E1 -15183.932,E2 -15183.932} C_VEL
LIN {X 0,Y 322.486,Z 335.752,A -85,B 0,C 180,E1 -15186.29,E2 -15186.29} C_VEL
LIN {X 0,Y 326.546,Z 366.119,A -85,B 0,C 180,E1 -15187.248,E2 -15187.248} C_VEL
LIN {X 0,Y 327.995,Z 379.009,A -85,B 0,C 180,E1 -15187.629,E2 -15187.629} C_VEL
LIN {X 0,Y 326.704,Z 444.893,A -85,B 0,C 180,E1 -15189.085,E2 -15189.085} C_VEL
LIN {X 0,Y 326.02,Z 458.084,A -85,B 0,C 180,E1 -15189.617,E2 -15189.617} C_VEL
LIN {X 0,Y 325.053,Z 470.214,A -85,B 0,C 180,E1 -15190.337,E2 -15190.337} C_VEL
LIN {X 0,Y 323.851,Z 482.455,A -85,B 0,C 180,E1 -15191.331,E2 -15191.331} C_VEL
LIN {X 0,Y 322.64,Z 494.086,A -85,B 0,C 180,E1 -15192.571,E2 -15192.571} C_VEL
LIN {X 0,Y 321.491,Z 504.931,A -85,B 0,C 180,E1 -15194.034,E2 -15194.034} C_VEL
LIN {X 0,Y 320.398,Z 514.79,A -85,B 0,C 180,E1 -15195.713,E2 -15195.713} C_VEL
LIN {X 0,Y 319.381,Z 523.748,A -85,B 0,C 180,E1 -15197.61,E2 -15197.61} C_VEL
LIN {X 0,Y 318.644,Z 530.925,A -85,B 0,C 180,E1 -15199.515,E2 -15199.515} C_VEL
LIN {X 0,Y 318.147,Z 537.463,A -85,B 0,C 180,E1 -15201.744,E2 -15201.744} C_VEL
LIN {X 0,Y 317.917,Z 541.767,A -85,B 0,C 180,E1 -15203.653,E2 -15203.653} C_VEL
LIN {X 0,Y 317.867,Z 544.045,A -85,B 0,C 180,E1 -15204.925,E2 -15204.925} C_VEL
LIN {X 0,Y 317.888,Z 545.854,A -85,B 0,C 180,E1 -15206.196,E2 -15206.196} C_VEL
LIN {X 0,Y 317.896,Z 548.166,A -85,B 0,C 180,E1 -15208.732,E2 -15208.732} C_VEL
LIN {X 0,Y 317.949,Z 548.73,A -85,B 0,C 180,E1 -15209.999,E2 -15209.999} C_VEL
LIN {X 0,Y 317.867,Z 548.863,A -85,B 0,C 180,E1 -15211.266,E2 -15211.266} C_VEL
LIN {X 0,Y 317.842,Z 547.92,A -85,B 0,C 180,E1 -15213.803,E2 -15213.803} C_VEL
LIN {X 0,Y 317.837,Z 546.163,A -85,B 0,C 180,E1 -15215.709,E2 -15215.709} C_VEL
LIN {X 0,Y 318.192,Z 542.378,A -85,B 0,C 180,E1 -15218.254,E2 -15218.254} C_VEL
LIN {X 0,Y 318.683,Z 538.328,A -85,B 0,C 180,E1 -15220.161,E2 -15220.161} C_VEL
LIN {X 0,Y 319.614,Z 532.133,A -85,B 0,C 180,E1 -15222.379,E2 -15222.379} C_VEL
LIN {X 0,Y 320.937,Z 525.413,A -85,B 0,C 180,E1 -15224.261,E2 -15224.261} C_VEL
LIN {X 0,Y 322.25,Z 517.565,A -85,B 0,C 180,E1 -15226.043,E2 -15226.043} C_VEL
LIN {X 0,Y 323.788,Z 508.595,A -85,B 0,C 180,E1 -15227.69,E2 -15227.69} C_VEL
LIN {X 0,Y 325.619,Z 498.118,A -85,B 0,C 180,E1 -15229.216,E2 -15229.216} C_VEL
LIN {X 0,Y 327.437,Z 486.351,A -85,B 0,C 180,E1 -15230.576,E2 -15230.576} C_VEL
LIN {X 0,Y 329.047,Z 474.531,A -85,B 0,C 180,E1 -15231.618,E2 -15231.618} C_VEL
LIN {X 0,Y 330.44,Z 462.262,A -85,B 0,C 180,E1 -15232.426,E2 -15232.426} C_VEL
LIN {X 0,Y 331.504,Z 449.716,A -85,B 0,C 180,E1 -15233.009,E2 -15233.009} C_VEL
LIN {X 0,Y 332.093,Z 436.856,A -85,B 0,C 180,E1 -15233.378,E2 -15233.378} C_VEL
LIN {X 0,Y 333.424,Z 378.176,A -85,B 0,C 180,E1 -15234.659,E2 -15234.659} C_VEL
LIN {X 0,Y 328.989,Z 352.144,A -85,B 0,C 180,E1 -15235.699,E2 -15235.699} C_VEL
LIN {X 0,Y 325.395,Z 334.872,A -85,B 0,C 180,E1 -15236.497,E2 -15236.497} C_VEL
LIN {X 0,Y 325.444,Z 331.385,A -85,B 0,C 180,E1 -15237.403,E2 -15237.403} C_VEL
LIN {X 0,Y 323.621,Z 322.424,A -85,B 0,C 180,E1 -15239.965,E2 -15239.965} C_VEL
LIN {X 0,Y 321.105,Z 311.807,A -85,B 0,C 180,E1 -15243.172,E2 -15243.172} C_VEL
LIN {X 0,Y 319.598,Z 305.68,A -85,B 0,C 180,E1 -15245.121,E2 -15245.121} C_VEL
LIN {X 0,Y 319.554,Z 305.681,A -85,B 0,C 180,E1 -15248.01,E2 -15248.01} C_VEL
LIN {X 0,Y 319.523,Z 305.68,A -85,B 0,C 180,E1 -15251.596,E2 -15251.596} C_VEL
LIN {X 0,Y 319.485,Z 305.688,A -85,B 0,C 180,E1 -15255.257,E2 -15255.257} C_VEL
LIN {X 0,Y 319.525,Z 305.68,A -85,B 0,C 180,E1 -15258.711,E2 -15258.711} C_VEL
LIN {X 0,Y 319.558,Z 305.674,A -85,B 0,C 180,E1 -15262.347,E2 -15262.347} C_VEL
LIN {X 0,Y 319.556,Z 305.672,A -85,B 0,C 180,E1 -15265.123,E2 -15265.123} C_VEL
LIN {X 0,Y 319.562,Z 305.674,A -85,B 0,C 180,E1 -15269.059,E2 -15269.059} C_VEL
LIN {X 0,Y 319.601,Z 305.667,A -85,B 0,C 180,E1 -15272.498,E2 -15272.498} C_VEL
LIN {X 0,Y 319.601,Z 305.665,A -85,B 0,C 180,E1 -15275.304,E2 -15275.304} C_VEL
LIN {X 0,Y 319.593,Z 305.673,A -85,B 0,C 180,E1 -15278.048,E2 -15278.048} C_VEL
LIN {X 0,Y 319.685,Z 305.663,A -85,B 0,C 180,E1 -15280.962,E2 -15280.962} C_VEL
LIN {X 0,Y 319.727,Z 305.658,A -85,B 0,C 180,E1 -15285.276,E2 -15285.276} C_VEL
LIN {X 0,Y 319.754,Z 305.653,A -85,B 0,C 180,E1 -15289.873,E2 -15289.873} C_VEL
LIN {X 0,Y 319.93,Z 305.625,A -85,B 0,C 180,E1 -15292.426,E2 -15292.426} C_VEL
LIN {X 0,Y 319.745,Z 305.654,A -85,B 0,C 180,E1 -15294.956,E2 -15294.956} C_VEL
LIN {X 0,Y 319.988,Z 305.624,A -85,B 0,C 180,E1 -15297.483,E2 -15297.483} C_VEL
LIN {X 0,Y 320.147,Z 305.6,A -85,B 0,C 180,E1 -15300,E2 -15300} C_VEL
LIN {X 0,Y 319.988,Z 305.624,A -85,B 0,C 180,E1 -15302.518,E2 -15302.518} C_VEL
LIN {X 0,Y 319.928,Z 305.627,A -85,B 0,C 180,E1 -15306.655,E2 -15306.655} C_VEL
LIN {X 0,Y 319.755,Z 305.649,A -85,B 0,C 180,E1 -15310.128,E2 -15310.128} C_VEL
LIN {X 0,Y 319.728,Z 305.655,A -85,B 0,C 180,E1 -15314.725,E2 -15314.725} C_VEL
LIN {X 0,Y 319.686,Z 305.663,A -85,B 0,C 180,E1 -15319.038,E2 -15319.038} C_VEL
LIN {X 0,Y 319.568,Z 305.68,A -85,B 0,C 180,E1 -15323.32,E2 -15323.32} C_VEL
LIN {X 0,Y 319.632,Z 305.667,A -85,B 0,C 180,E1 -15326.089,E2 -15326.089} C_VEL
LIN {X 0,Y 319.577,Z 305.672,A -85,B 0,C 180,E1 -15328.935,E2 -15328.935} C_VEL
LIN {X 0,Y 319.529,Z 305.676,A -85,B 0,C 180,E1 -15331.863,E2 -15331.863} C_VEL
LIN {X 0,Y 319.577,Z 305.671,A -85,B 0,C 180,E1 -15335.544,E2 -15335.544} C_VEL
LIN {X 0,Y 319.557,Z 305.679,A -85,B 0,C 180,E1 -15339.67,E2 -15339.67} C_VEL
LIN {X 0,Y 319.52,Z 305.682,A -85,B 0,C 180,E1 -15343.461,E2 -15343.461} C_VEL
LIN {X 0,Y 319.551,Z 305.682,A -85,B 0,C 180,E1 -15347.017,E2 -15347.017} C_VEL
LIN {X 0,Y 319.544,Z 305.682,A -85,B 0,C 180,E1 -15350.372,E2 -15350.372} C_VEL
LIN {X 0,Y 319.618,Z 305.837,A -85,B 0,C 180,E1 -15352.992,E2 -15352.992} C_VEL
LIN {X 0,Y 320.475,Z 309.09,A -85,B 0,C 180,E1 -15354.05,E2 -15354.05} C_VEL
LIN {X 0,Y 329.289,Z 327.608,A -85,B 0,C 180,E1 -15355.413,E2 -15355.413} C_VEL
LIN {X 0,Y 334.48,Z 339.89,A -85,B 0,C 180,E1 -15356.204,E2 -15356.204} C_VEL
LIN {X 0,Y 332.334,Z 415.942,A -85,B 0,C 180,E1 -15357.859,E2 -15357.859} C_VEL
LIN {X 0,Y 331.682,Z 429.59,A -85,B 0,C 180,E1 -15358.416,E2 -15358.416} C_VEL
LIN {X 0,Y 330.587,Z 441.903,A -85,B 0,C 180,E1 -15359.145,E2 -15359.145} C_VEL
LIN {X 0,Y 329.305,Z 453.433,A -85,B 0,C 180,E1 -15360.076,E2 -15360.076} C_VEL
LIN {X 0,Y 327.954,Z 464.475,A -85,B 0,C 180,E1 -15361.244,E2 -15361.244} C_VEL
LIN {X 0,Y 326.342,Z 474.745,A -85,B 0,C 180,E1 -15362.593,E2 -15362.593} C_VEL
LIN {X 0,Y 324.892,Z 483.523,A -85,B 0,C 180,E1 -15364.022,E2 -15364.022} C_VEL
LIN {X 0,Y 323.456,Z 491.56,A -85,B 0,C 180,E1 -15365.618,E2 -15365.618} C_VEL
LIN {X 0,Y 321.915,Z 499.344,A -85,B 0,C 180,E1 -15367.54,E2 -15367.54} C_VEL
LIN {X 0,Y 320.688,Z 505.544,A -85,B 0,C 180,E1 -15369.474,E2 -15369.474} C_VEL
LIN {X 0,Y 319.688,Z 510.489,A -85,B 0,C 180,E1 -15371.442,E2 -15371.442} C_VEL
LIN {X 0,Y 318.981,Z 514.146,A -85,B 0,C 180,E1 -15373.357,E2 -15373.357} C_VEL
LIN {X 0,Y 318.638,Z 516.051,A -85,B 0,C 180,E1 -15374.653,E2 -15374.653} C_VEL
LIN {X 0,Y 318.302,Z 517.794,A -85,B 0,C 180,E1 -15376.292,E2 -15376.292} C_VEL
LIN {X 0,Y 317.936,Z 519.119,A -85,B 0,C 180,E1 -15378.526,E2 -15378.526} C_VEL
LIN {X 0,Y 317.814,Z 519.347,A -85,B 0,C 180,E1 -15379.811,E2 -15379.811} C_VEL
LIN {X 0,Y 317.82,Z 519.139,A -85,B 0,C 180,E1 -15381.096,E2 -15381.096} C_VEL
LIN {X 0,Y 317.898,Z 518.527,A -85,B 0,C 180,E1 -15382.378,E2 -15382.378} C_VEL
LIN {X 0,Y 318.029,Z 517.254,A -85,B 0,C 180,E1 -15383.96,E2 -15383.96} C_VEL
LIN {X 0,Y 318.137,Z 514.305,A -85,B 0,C 180,E1 -15386.201,E2 -15386.201} C_VEL
LIN {X 0,Y 318.518,Z 510.722,A -85,B 0,C 180,E1 -15388.104,E2 -15388.104} C_VEL
LIN {X 0,Y 318.911,Z 506.053,A -85,B 0,C 180,E1 -15390.001,E2 -15390.001} C_VEL
LIN {X 0,Y 319.779,Z 499.023,A -85,B 0,C 180,E1 -15392.205,E2 -15392.205} C_VEL
LIN {X 0,Y 320.705,Z 491.407,A -85,B 0,C 180,E1 -15394.085,E2 -15394.085} C_VEL
LIN {X 0,Y 321.784,Z 481.856,A -85,B 0,C 180,E1 -15395.956,E2 -15395.956} C_VEL
LIN {X 0,Y 322.968,Z 471.992,A -85,B 0,C 180,E1 -15397.503,E2 -15397.503} C_VEL
LIN {X 0,Y 324.135,Z 460.874,A -85,B 0,C 180,E1 -15398.888,E2 -15398.888} C_VEL
LIN {X 0,Y 325.104,Z 450.003,A -85,B 0,C 180,E1 -15399.96,E2 -15399.96} C_VEL
LIN {X 0,Y 325.903,Z 438.018,A -85,B 0,C 180,E1 -15400.877,E2 -15400.877} C_VEL
LIN {X 0,Y 326.648,Z 425.586,A -85,B 0,C 180,E1 -15401.559,E2 -15401.559} C_VEL
LIN {X 0,Y 327.037,Z 412.725,A -85,B 0,C 180,E1 -15402.017,E2 -15402.017} C_VEL
LIN {X 0,Y 328.65,Z 334.793,A -85,B 0,C 180,E1 -15403.707,E2 -15403.707} C_VEL
LIN {X 0,Y 327.071,Z 327.696,A -85,B 0,C 180,E1 -15403.97,E2 -15403.97} C_VEL
LIN {X 0,Y 320.248,Z 308.163,A -85,B 0,C 180,E1 -15404.907,E2 -15404.907} C_VEL
LIN {X 0,Y 319.691,Z 305.661,A -85,B 0,C 180,E1 -15405.705,E2 -15405.705} C_VEL
LIN {X 0,Y 319.634,Z 305.669,A -85,B 0,C 180,E1 -15409.258,E2 -15409.258} C_VEL
LIN {X 0,Y 319.556,Z 305.676,A -85,B 0,C 180,E1 -15413.321,E2 -15413.321} C_VEL
LIN {X 0,Y 319.572,Z 305.672,A -85,B 0,C 180,E1 -15416.094,E2 -15416.094} C_VEL
LIN {X 0,Y 319.546,Z 305.683,A -85,B 0,C 180,E1 -15418.939,E2 -15418.939} C_VEL
LIN {X 0,Y 319.529,Z 305.68,A -85,B 0,C 180,E1 -15421.863,E2 -15421.863} C_VEL
LIN {X 0,Y 319.585,Z 305.675,A -85,B 0,C 180,E1 -15425.543,E2 -15425.543} C_VEL
LIN {X 0,Y 319.538,Z 305.678,A -85,B 0,C 180,E1 -15427.075,E2 -15427.075} C_VEL
LIN {X 0,Y 318.879,Z 305.762,A -85,B 0,C 180,E1 -15428.127,E2 -15428.127} C_VEL
LIN {X 0,Y 316.043,Z 306.118,A -85,B 0,C 180,E1 -15429.84,E2 -15429.84} C_VEL
LIN {X 0,Y 313.619,Z 306.419,A -85,B 0,C 180,E1 -15431.228,E2 -15431.228} C_VEL
LIN {X 0,Y 312.554,Z 306.548,A -85,B 0,C 180,E1 -15432.303,E2 -15432.303} C_VEL
LIN {X 0,Y 312.454,Z 306.558,A -85,B 0,C 180,E1 -15432.667,E2 -15432.667} C_VEL
LIN {X 0,Y 312.462,Z 306.559,A -85,B 0,C 180,E1 -15436.035,E2 -15436.035} C_VEL
LIN {X 0,Y 312.46,Z 306.562,A -85,B 0,C 180,E1 -15439.886,E2 -15439.886} C_VEL
LIN {X 0,Y 312.538,Z 306.549,A -85,B 0,C 180,E1 -15444.051,E2 -15444.051} C_VEL
LIN {X 0,Y 312.506,Z 306.555,A -85,B 0,C 180,E1 -15447.333,E2 -15447.333} C_VEL
LIN {X 0,Y 312.511,Z 306.556,A -85,B 0,C 180,E1 -15451.292,E2 -15451.292} C_VEL
LIN {X 0,Y 312.53,Z 306.545,A -85,B 0,C 180,E1 -15454.706,E2 -15454.706} C_VEL
LIN {X 0,Y 312.545,Z 306.551,A -85,B 0,C 180,E1 -15457.525,E2 -15457.525} C_VEL
LIN {X 0,Y 312.587,Z 306.548,A -85,B 0,C 180,E1 -15461.653,E2 -15461.653} C_VEL
LIN {X 0,Y 312.691,Z 306.528,A -85,B 0,C 180,E1 -15465.686,E2 -15465.686} C_VEL
LIN {X 0,Y 312.689,Z 306.533,A -85,B 0,C 180,E1 -15469.641,E2 -15469.641} C_VEL
LIN {X 0,Y 312.801,Z 306.52,A -85,B 0,C 180,E1 -15472.252,E2 -15472.252} C_VEL
LIN {X 0,Y 312.692,Z 306.526,A -85,B 0,C 180,E1 -15474.842,E2 -15474.842} C_VEL
LIN {X 0,Y 312.971,Z 306.498,A -85,B 0,C 180,E1 -15478.713,E2 -15478.713} C_VEL
LIN {X 0,Y 312.98,Z 306.495,A -85,B 0,C 180,E1 -15481.286,E2 -15481.286} C_VEL
LIN {X 0,Y 312.843,Z 306.512,A -85,B 0,C 180,E1 -15486.449,E2 -15486.449} C_VEL
LIN {X 0,Y 312.754,Z 306.524,A -85,B 0,C 180,E1 -15489.05,E2 -15489.05} C_VEL
LIN {X 0,Y 312.636,Z 306.54,A -85,B 0,C 180,E1 -15492.991,E2 -15492.991} C_VEL
LIN {X 0,Y 312.625,Z 306.54,A -85,B 0,C 180,E1 -15495.65,E2 -15495.65} C_VEL
LIN {X 0,Y 312.542,Z 306.55,A -85,B 0,C 180,E1 -15499.712,E2 -15499.712} C_VEL
LIN {X 0,Y 312.525,Z 306.557,A -85,B 0,C 180,E1 -15502.778,E2 -15502.778} C_VEL
LIN {X 0,Y 312.531,Z 306.552,A -85,B 0,C 180,E1 -15505.906,E2 -15505.906} C_VEL
LIN {X 0,Y 312.475,Z 306.56,A -85,B 0,C 180,E1 -15509.657,E2 -15509.657} C_VEL
LIN {X 0,Y 312.523,Z 306.554,A -85,B 0,C 180,E1 -15513.688,E2 -15513.688} C_VEL
LIN {X 0,Y 312.516,Z 306.557,A -85,B 0,C 180,E1 -15517.386,E2 -15517.386} C_VEL
LIN {X 0,Y 312.443,Z 306.565,A -85,B 0,C 180,E1 -15520.716,E2 -15520.716} C_VEL
LIN {X 0,Y 312.452,Z 306.562,A -85,B 0,C 180,E1 -15524.209,E2 -15524.209} C_VEL
LIN {X 0,Y 312.457,Z 306.562,A -85,B 0,C 180,E1 -15527.924,E2 -15527.924} C_VEL
LIN {X 0,Y 312.486,Z 306.56,A -85,B 0,C 180,E1 -15531.922,E2 -15531.922} C_VEL
LIN {X 0,Y 312.532,Z 306.554,A -85,B 0,C 180,E1 -15534.219,E2 -15534.219} C_VEL
LIN {X 0,Y 312.552,Z 306.602,A -85,B 0,C 180,E1 -15538.118,E2 -15538.118} C_VEL
LIN {X 0,Y 314.955,Z 318,A -85,B 0,C 180,E1 -15541.33,E2 -15541.33} C_VEL
LIN {X 0,Y 316.462,Z 326.51,A -85,B 0,C 180,E1 -15543.629,E2 -15543.629} C_VEL
LIN {X 0,Y 315.684,Z 334.744,A -85,B 0,C 180,E1 -15545.677,E2 -15545.677} C_VEL
LIN {X 0,Y 315.633,Z 335.341,A -85,B 0,C 180,E1 -15545.825,E2 -15545.825} C_VEL
LIN {X 0,Y 319.895,Z 367.256,A -85,B 0,C 180,E1 -15546.86,E2 -15546.86} C_VEL
LIN {X 0,Y 321.279,Z 379.663,A -85,B 0,C 180,E1 -15547.236,E2 -15547.236} C_VEL
LIN {X 0,Y 319.952,Z 444.765,A -85,B 0,C 180,E1 -15548.707,E2 -15548.707} C_VEL
LIN {X 0,Y 319.126,Z 458.643,A -85,B 0,C 180,E1 -15549.283,E2 -15549.283} C_VEL
LIN {X 0,Y 318.156,Z 471.091,A -85,B 0,C 180,E1 -15550.061,E2 -15550.061} C_VEL
LIN {X 0,Y 316.917,Z 483,A -85,B 0,C 180,E1 -15551.074,E2 -15551.074} C_VEL
LIN {X 0,Y 315.674,Z 494.473,A -85,B 0,C 180,E1 -15552.341,E2 -15552.341} C_VEL
LIN {X 0,Y 314.559,Z 504.702,A -85,B 0,C 180,E1 -15553.763,E2 -15553.763} C_VEL
LIN {X 0,Y 313.5,Z 514.094,A -85,B 0,C 180,E1 -15555.391,E2 -15555.391} C_VEL
LIN {X 0,Y 312.41,Z 523.112,A -85,B 0,C 180,E1 -15557.329,E2 -15557.329} C_VEL
LIN {X 0,Y 311.616,Z 530.359,A -85,B 0,C 180,E1 -15559.276,E2 -15559.276} C_VEL
LIN {X 0,Y 311.181,Z 535.246,A -85,B 0,C 180,E1 -15560.903,E2 -15560.903} C_VEL
LIN {X 0,Y 310.912,Z 539.988,A -85,B 0,C 180,E1 -15562.857,E2 -15562.857} C_VEL
LIN {X 0,Y 310.783,Z 543.595,A -85,B 0,C 180,E1 -15564.809,E2 -15564.809} C_VEL
LIN {X 0,Y 310.794,Z 545.441,A -85,B 0,C 180,E1 -15566.109,E2 -15566.109} C_VEL
LIN {X 0,Y 310.763,Z 546.815,A -85,B 0,C 180,E1 -15567.407,E2 -15567.407} C_VEL
LIN {X 0,Y 310.802,Z 547.791,A -85,B 0,C 180,E1 -15568.703,E2 -15568.703} C_VEL
LIN {X 0,Y 310.857,Z 548.373,A -85,B 0,C 180,E1 -15569.999,E2 -15569.999} C_VEL
LIN {X 0,Y 310.774,Z 548.54,A -85,B 0,C 180,E1 -15571.295,E2 -15571.295} C_VEL
LIN {X 0,Y 310.749,Z 547.633,A -85,B 0,C 180,E1 -15573.89,E2 -15573.89} C_VEL
LIN {X 0,Y 310.817,Z 545.156,A -85,B 0,C 180,E1 -15576.491,E2 -15576.491} C_VEL
LIN {X 0,Y 311.135,Z 542.172,A -85,B 0,C 180,E1 -15578.442,E2 -15578.442} C_VEL
LIN {X 0,Y 311.659,Z 538.16,A -85,B 0,C 180,E1 -15580.392,E2 -15580.392} C_VEL
LIN {X 0,Y 312.658,Z 532.029,A -85,B 0,C 180,E1 -15582.659,E2 -15582.659} C_VEL
LIN {X 0,Y 314.054,Z 525.363,A -85,B 0,C 180,E1 -15584.581,E2 -15584.581} C_VEL
LIN {X 0,Y 315.519,Z 517,A -85,B 0,C 180,E1 -15586.524,E2 -15586.524} C_VEL
LIN {X 0,Y 317.022,Z 508.697,A -85,B 0,C 180,E1 -15588.08,E2 -15588.08} C_VEL
LIN {X 0,Y 318.915,Z 498.33,A -85,B 0,C 180,E1 -15589.637,E2 -15589.637} C_VEL
LIN {X 0,Y 320.826,Z 486.68,A -85,B 0,C 180,E1 -15591.02,E2 -15591.02} C_VEL
LIN {X 0,Y 322.496,Z 475.118,A -85,B 0,C 180,E1 -15592.08,E2 -15592.08} C_VEL
LIN {X 0,Y 323.933,Z 463.131,A -85,B 0,C 180,E1 -15592.902,E2 -15592.902} C_VEL
LIN {X 0,Y 325.098,Z 450.163,A -85,B 0,C 180,E1 -15593.531,E2 -15593.531} C_VEL
LIN {X 0,Y 325.773,Z 436.279,A -85,B 0,C 180,E1 -15593.943,E2 -15593.943} C_VEL
LIN {X 0,Y 327.198,Z 380.035,A -85,B 0,C 180,E1 -15595.185,E2 -15595.185} C_VEL
LIN {X 0,Y 323.556,Z 357.493,A -85,B 0,C 180,E1 -15596.093,E2 -15596.093} C_VEL
LIN {X 0,Y 319.194,Z 336.552,A -85,B 0,C 180,E1 -15597.065,E2 -15597.065} C_VEL
LIN {X 0,Y 318.734,Z 334.465,A -85,B 0,C 180,E1 -15597.199,E2 -15597.199} C_VEL
LIN {X 0,Y 317.336,Z 326.526,A -85,B 0,C 180,E1 -15599.485,E2 -15599.485} C_VEL
LIN {X 0,Y 314.506,Z 314.455,A -85,B 0,C 180,E1 -15603.193,E2 -15603.193} C_VEL
LIN {X 0,Y 312.529,Z 306.558,A -85,B 0,C 180,E1 -15605.779,E2 -15605.779} C_VEL
LIN {X 0,Y 312.5,Z 306.557,A -85,B 0,C 180,E1 -15609.028,E2 -15609.028} C_VEL
LIN {X 0,Y 312.487,Z 306.562,A -85,B 0,C 180,E1 -15612.431,E2 -15612.431} C_VEL
LIN {X 0,Y 312.455,Z 306.562,A -85,B 0,C 180,E1 -15616.034,E2 -15616.034} C_VEL
LIN {X 0,Y 312.5,Z 306.555,A -85,B 0,C 180,E1 -15619.874,E2 -15619.874} C_VEL
LIN {X 0,Y 312.532,Z 306.554,A -85,B 0,C 180,E1 -15624.05,E2 -15624.05} C_VEL
LIN {X 0,Y 312.5,Z 306.555,A -85,B 0,C 180,E1 -15627.333,E2 -15627.333} C_VEL
LIN {X 0,Y 312.54,Z 306.547,A -85,B 0,C 180,E1 -15631.279,E2 -15631.279} C_VEL
LIN {X 0,Y 312.581,Z 306.544,A -85,B 0,C 180,E1 -15634.711,E2 -15634.711} C_VEL
LIN {X 0,Y 312.583,Z 306.546,A -85,B 0,C 180,E1 -15637.529,E2 -15637.529} C_VEL
LIN {X 0,Y 312.634,Z 306.54,A -85,B 0,C 180,E1 -15641.656,E2 -15641.656} C_VEL
LIN {X 0,Y 312.69,Z 306.534,A -85,B 0,C 180,E1 -15645.686,E2 -15645.686} C_VEL
LIN {X 0,Y 312.698,Z 306.533,A -85,B 0,C 180,E1 -15649.642,E2 -15649.642} C_VEL
LIN {X 0,Y 312.868,Z 306.504,A -85,B 0,C 180,E1 -15652.254,E2 -15652.254} C_VEL
LIN {X 0,Y 312.715,Z 306.531,A -85,B 0,C 180,E1 -15654.843,E2 -15654.843} C_VEL
LIN {X 0,Y 312.987,Z 306.499,A -85,B 0,C 180,E1 -15658.714,E2 -15658.714} C_VEL
LIN {X 0,Y 312.987,Z 306.493,A -85,B 0,C 180,E1 -15661.287,E2 -15661.287} C_VEL
LIN {X 0,Y 312.714,Z 306.525,A -85,B 0,C 180,E1 -15665.158,E2 -15665.158} C_VEL
LIN {X 0,Y 312.869,Z 306.509,A -85,B 0,C 180,E1 -15667.746,E2 -15667.746} C_VEL
LIN {X 0,Y 312.666,Z 306.535,A -85,B 0,C 180,E1 -15671.672,E2 -15671.672} C_VEL
LIN {X 0,Y 312.697,Z 306.532,A -85,B 0,C 180,E1 -15674.888,E2 -15674.888} C_VEL
LIN {X 0,Y 312.627,Z 306.545,A -85,B 0,C 180,E1 -15679.237,E2 -15679.237} C_VEL
LIN {X 0,Y 312.543,Z 306.551,A -85,B 0,C 180,E1 -15682.79,E2 -15682.79} C_VEL
LIN {X 0,Y 312.6,Z 306.543,A -85,B 0,C 180,E1 -15685.936,E2 -15685.936} C_VEL
LIN {X 0,Y 312.536,Z 306.551,A -85,B 0,C 180,E1 -15689.652,E2 -15689.652} C_VEL
LIN {X 0,Y 312.517,Z 306.555,A -85,B 0,C 180,E1 -15693.69,E2 -15693.69} C_VEL
LIN {X 0,Y 312.513,Z 306.554,A -85,B 0,C 180,E1 -15697.388,E2 -15697.388} C_VEL
LIN {X 0,Y 312.486,Z 306.557,A -85,B 0,C 180,E1 -15700.71,E2 -15700.71} C_VEL
LIN {X 0,Y 312.45,Z 306.565,A -85,B 0,C 180,E1 -15704.211,E2 -15704.211} C_VEL
LIN {X 0,Y 312.454,Z 306.563,A -85,B 0,C 180,E1 -15707.926,E2 -15707.926} C_VEL
LIN {X 0,Y 312.515,Z 306.557,A -85,B 0,C 180,E1 -15712.273,E2 -15712.273} C_VEL
LIN {X 0,Y 313.292,Z 309.496,A -85,B 0,C 180,E1 -15713.277,E2 -15713.277} C_VEL
LIN {X 0,Y 322.822,Z 329.039,A -85,B 0,C 180,E1 -15714.802,E2 -15714.802} C_VEL
LIN {X 0,Y 328.244,Z 341.74,A -85,B 0,C 180,E1 -15715.659,E2 -15715.659} C_VEL
LIN {X 0,Y 325.983,Z 416.617,A -85,B 0,C 180,E1 -15717.315,E2 -15717.315} C_VEL
LIN {X 0,Y 325.344,Z 429.775,A -85,B 0,C 180,E1 -15717.864,E2 -15717.864} C_VEL
LIN {X 0,Y 324.136,Z 442.698,A -85,B 0,C 180,E1 -15718.644,E2 -15718.644} C_VEL
LIN {X 0,Y 322.801,Z 454.091,A -85,B 0,C 180,E1 -15719.59,E2 -15719.59} C_VEL
LIN {X 0,Y 321.408,Z 464.941,A -85,B 0,C 180,E1 -15720.763,E2 -15720.763} C_VEL
LIN {X 0,Y 319.705,Z 475.33,A -85,B 0,C 180,E1 -15722.158,E2 -15722.158} C_VEL
LIN {X 0,Y 318.041,Z 484.928,A -85,B 0,C 180,E1 -15723.772,E2 -15723.772} C_VEL
LIN {X 0,Y 316.306,Z 493.778,A -85,B 0,C 180,E1 -15725.642,E2 -15725.642} C_VEL
LIN {X 0,Y 314.699,Z 501.484,A -85,B 0,C 180,E1 -15727.689,E2 -15727.689} C_VEL
LIN {X 0,Y 313.484,Z 507.328,A -85,B 0,C 180,E1 -15729.667,E2 -15729.667} C_VEL
LIN {X 0,Y 312.543,Z 511.881,A -85,B 0,C 180,E1 -15731.651,E2 -15731.651} C_VEL
LIN {X 0,Y 312.019,Z 514.263,A -85,B 0,C 180,E1 -15732.974,E2 -15732.974} C_VEL
LIN {X 0,Y 311.645,Z 516.203,A -85,B 0,C 180,E1 -15734.3,E2 -15734.3} C_VEL
LIN {X 0,Y 311.239,Z 518.171,A -85,B 0,C 180,E1 -15736.164,E2 -15736.164} C_VEL
LIN {X 0,Y 310.884,Z 519.404,A -85,B 0,C 180,E1 -15738.262,E2 -15738.262} C_VEL
LIN {X 0,Y 310.733,Z 519.664,A -85,B 0,C 180,E1 -15739.576,E2 -15739.576} C_VEL
LIN {X 0,Y 310.738,Z 519.519,A -85,B 0,C 180,E1 -15740.891,E2 -15740.891} C_VEL
LIN {X 0,Y 310.787,Z 518.942,A -85,B 0,C 180,E1 -15742.203,E2 -15742.203} C_VEL
LIN {X 0,Y 310.949,Z 517.555,A -85,B 0,C 180,E1 -15743.982,E2 -15743.982} C_VEL
LIN {X 0,Y 311.127,Z 513.787,A -85,B 0,C 180,E1 -15746.763,E2 -15746.763} C_VEL
LIN {X 0,Y 311.541,Z 509.922,A -85,B 0,C 180,E1 -15748.708,E2 -15748.708} C_VEL
LIN {X 0,Y 312.02,Z 504.947,A -85,B 0,C 180,E1 -15750.646,E2 -15750.646} C_VEL
LIN {X 0,Y 312.835,Z 498.688,A -85,B 0,C 180,E1 -15752.576,E2 -15752.576} C_VEL
LIN {X 0,Y 313.83,Z 490.858,A -85,B 0,C 180,E1 -15754.496,E2 -15754.496} C_VEL
LIN {X 0,Y 314.768,Z 482.895,A -85,B 0,C 180,E1 -15756.089,E2 -15756.089} C_VEL
LIN {X 0,Y 315.978,Z 473.172,A -85,B 0,C 180,E1 -15757.67,E2 -15757.67} C_VEL
LIN {X 0,Y 317.151,Z 462.339,A -85,B 0,C 180,E1 -15759.085,E2 -15759.085} C_VEL
LIN {X 0,Y 318.191,Z 451.726,A -85,B 0,C 180,E1 -15760.178,E2 -15760.178} C_VEL
LIN {X 0,Y 319.073,Z 439.013,A -85,B 0,C 180,E1 -15761.193,E2 -15761.193} C_VEL
LIN {X 0,Y 319.887,Z 426.082,A -85,B 0,C 180,E1 -15761.927,E2 -15761.927} C_VEL
LIN {X 0,Y 320.303,Z 413.32,A -85,B 0,C 180,E1 -15762.394,E2 -15762.394} C_VEL
LIN {X 0,Y 321.96,Z 335.624,A -85,B 0,C 180,E1 -15764.115,E2 -15764.115} C_VEL
LIN {X 0,Y 320.364,Z 329.019,A -85,B 0,C 180,E1 -15764.375,E2 -15764.375} C_VEL
LIN {X 0,Y 313.867,Z 310.778,A -85,B 0,C 180,E1 -15765.256,E2 -15765.256} C_VEL
LIN {X 0,Y 313.058,Z 308.548,A -85,B 0,C 180,E1 -15765.39,E2 -15765.39} C_VEL
LIN {X 0,Y 312.651,Z 306.54,A -85,B 0,C 180,E1 -15766.068,E2 -15766.068} C_VEL
LIN {X 0,Y 312.564,Z 306.548,A -85,B 0,C 180,E1 -15769.712,E2 -15769.712} C_VEL
LIN {X 0,Y 312.527,Z 306.556,A -85,B 0,C 180,E1 -15772.779,E2 -15772.779} C_VEL
LIN {X 0,Y 312.533,Z 306.549,A -85,B 0,C 180,E1 -15775.907,E2 -15775.907} C_VEL
LIN {X 0,Y 312.5,Z 306.556,A -85,B 0,C 180,E1 -15779.656,E2 -15779.656} C_VEL
LIN {X 0,Y 312.525,Z 306.553,A -85,B 0,C 180,E1 -15783.689,E2 -15783.689} C_VEL
LIN {X 0,Y 312.519,Z 306.557,A -85,B 0,C 180,E1 -15787.387,E2 -15787.387} C_VEL
LIN {X 0,Y 312.446,Z 306.562,A -85,B 0,C 180,E1 -15790.717,E2 -15790.717} C_VEL
LIN {X 0,Y 312.454,Z 306.558,A -85,B 0,C 180,E1 -15792.667,E2 -15792.667} C_VEL
LIN {X 0,Y 311.76,Z 306.65,A -85,B 0,C 180,E1 -15793.744,E2 -15793.744} C_VEL
LIN {X 0,Y 308.926,Z 307.002,A -85,B 0,C 180,E1 -15795.497,E2 -15795.497} C_VEL
LIN {X 0,Y 306.535,Z 307.298,A -85,B 0,C 180,E1 -15796.918,E2 -15796.918} C_VEL
LIN {X 0,Y 305.497,Z 307.426,A -85,B 0,C 180,E1 -15798.018,E2 -15798.018} C_VEL
LIN {X 0,Y 305.404,Z 307.436,A -85,B 0,C 180,E1 -15798.391,E2 -15798.391} C_VEL
LIN {X 0,Y 305.451,Z 307.437,A -85,B 0,C 180,E1 -15801.593,E2 -15801.593} C_VEL
LIN {X 0,Y 305.466,Z 307.428,A -85,B 0,C 180,E1 -15804.887,E2 -15804.887} C_VEL
LIN {X 0,Y 305.446,Z 307.434,A -85,B 0,C 180,E1 -15808.358,E2 -15808.358} C_VEL
LIN {X 0,Y 305.481,Z 307.431,A -85,B 0,C 180,E1 -15811.109,E2 -15811.109} C_VEL
LIN {X 0,Y 305.486,Z 307.424,A -85,B 0,C 180,E1 -15814.08,E2 -15814.08} C_VEL
LIN {X 0,Y 305.47,Z 307.432,A -85,B 0,C 180,E1 -15818.4,E2 -15818.4} C_VEL
LIN {X 0,Y 305.548,Z 307.422,A -85,B 0,C 180,E1 -15821.214,E2 -15821.214} C_VEL
LIN {X 0,Y 305.632,Z 307.404,A -85,B 0,C 180,E1 -15825.348,E2 -15825.348} C_VEL
LIN {X 0,Y 305.628,Z 307.412,A -85,B 0,C 180,E1 -15829.399,E2 -15829.399} C_VEL
LIN {X 0,Y 305.751,Z 307.4,A -85,B 0,C 180,E1 -15832.072,E2 -15832.072} C_VEL
LIN {X 0,Y 305.662,Z 307.401,A -85,B 0,C 180,E1 -15834.723,E2 -15834.723} C_VEL
LIN {X 0,Y 305.939,Z 307.374,A -85,B 0,C 180,E1 -15838.683,E2 -15838.683} C_VEL
LIN {X 0,Y 305.947,Z 307.371,A -85,B 0,C 180,E1 -15841.316,E2 -15841.316} C_VEL
LIN {X 0,Y 305.788,Z 307.389,A -85,B 0,C 180,E1 -15846.598,E2 -15846.598} C_VEL
LIN {X 0,Y 305.698,Z 307.402,A -85,B 0,C 180,E1 -15849.261,E2 -15849.261} C_VEL
LIN {X 0,Y 305.589,Z 307.416,A -85,B 0,C 180,E1 -15853.296,E2 -15853.296} C_VEL
LIN {X 0,Y 305.554,Z 307.422,A -85,B 0,C 180,E1 -15856.022,E2 -15856.022} C_VEL
LIN {X 0,Y 305.487,Z 307.43,A -85,B 0,C 180,E1 -15860.187,E2 -15860.187} C_VEL
LIN {X 0,Y 305.477,Z 307.433,A -85,B 0,C 180,E1 -15864.464,E2 -15864.464} C_VEL
LIN {X 0,Y 305.457,Z 307.435,A -85,B 0,C 180,E1 -15867.397,E2 -15867.397} C_VEL
LIN {X 0,Y 305.421,Z 307.439,A -85,B 0,C 180,E1 -15870.413,E2 -15870.413} C_VEL
LIN {X 0,Y 305.467,Z 307.432,A -85,B 0,C 180,E1 -15874.078,E2 -15874.078} C_VEL
LIN {X 0,Y 305.456,Z 307.436,A -85,B 0,C 180,E1 -15876.742,E2 -15876.742} C_VEL
